// TwinCAT 3 PLC project PLCIO
// ProgramVersion: 3.1.4024.0
// libraries:
//   Tc2_ControllerToolbox, * (Beckhoff Automation GmbH)
//   Tc2_IoFunctions, * (Beckhoff Automation GmbH)
//   Tc2_ModbusRTU, * (Beckhoff Automation GmbH)
//   Tc2_ModbusSrv, * (Beckhoff Automation GmbH)
//   Tc2_SerialCom, * (Beckhoff Automation GmbH)
//   Tc2_Standard, * (Beckhoff Automation GmbH)
//   Tc2_System, * (Beckhoff Automation GmbH)
//   Tc2_TempController, * (Beckhoff Automation GmbH)
//   Tc2_Utilities, * (Beckhoff Automation GmbH)
//   Tc3_EventLogger, * (Beckhoff Automation GmbH)
//   Tc3_Module, * (Beckhoff Automation GmbH)
// project tree:
//   DUTs/ ST_CSV_Record.TcDUT, ST_Recipe1.TcDUT, ST_Array.TcDUT
//   GVLs/ GVL.TcGVL, GVL_CMD.TcGVL (not stored), GVL_COM.TcGVL, GVL_IO.TcGVL (not stored), GVL_OP_A.TcGVL (not stored), GVL_OP_D.TcGVL (not stored), GVL_P2P.TcGVL (not stored), GVL_Recipe.TcGVL
//   / PlcTask.TcTTO, RecipeManager.TcRMO (not stored)
//   POUs/CSV read_write in binary mode/ P_BinaryModeRead.TcPOU, P_BinaryModeWrite.TcPOU
//   POUs/CSV read_write in text mode/ P_TextModeRead.TcPOU, P_TextModeWrite.TcPOU
//   POUs/ Convert2Csv.TcPOU, MAIN.TcPOU, P_ArgToConvExample.TcPOU, P_StringToConvExample.TcPOU, RecipeHandler.TcPOU, TextFieldInputHandler.TcPOU, VisuInit.TcPOU
//   POUs/FunctionBlock/ FB_AI_STATUS_Check.TcPOU, FB_AVG10.TcPOU, FB_DeviationCheck.TcPOU, FB_NoiseCheck.TcPOU, FB_PID.TcPOU, FB_Ramp2.TcPOU, FB_RampControl.TcPOU, FB_Ramp_0.TcPOU, FB_RcpRamp.TcPOU
//   POUs/Function/ F_ET2Sec.TcPOU, F_Int2Real.TcPOU, F_LH_PV.TcPOU, F_LH_SV.TcPOU, F_OPSTATE.TcPOU, F_TB_PV2REAL.TcPOU, F_TB_Rx_BCC.TcPOU, F_TB_SV2STR.TcPOU, F_TB_Tx_BCC.TcPOU
//   POUs/MR_PRG/ P00_Main.TcPOU, P00_OP.TcPOU, P01_Init_N_Retain.TcPOU, P02_Init_MC.TcPOU, P11_Rx_TV.TcPOU, P12_Rx_IH.TcPOU, P13_DI_N_Check.TcPOU, P15_AI.TcPOU, P21_AL_WN.TcPOU, P22_RCP_Ctrl.TcPOU, P24_Rot_Calibration.TcPOU, P25_US_Ctrl.TcPOU, P31_BypassV.TcPOU, P41_DOR_VAC.TcPOU, P41_DOR_VAC_Check.TcPOU, P42_DOR_ATM.TcPOU, P43_SH_UpDw.TcPOU, P49_MO_SRC.TcPOU, P53_DO_VV.TcPOU, P54_DO_ETC.TcPOU, P61_AO.TcPOU, P62_Tx_TV.TcPOU, P63_Tx_IH.TcPOU, REF_P02_KL1501.TcPOU
//   POUs/P02_P2P/ P00_Task_Fast.TcPOU, P02_P2P.TcPOU, P2P_LH.TcPOU, P2P_TB.TcPOU, Task_Fast_LH.TcPOU, Task_Fast_TB.TcPOU
// real-time tasks:
//   TASK PlcTask: cycle T#10ms, priority 20, ADS port 350
//   TASK PlcRecipe: cycle T#10ms, priority 1, ADS port 351

CONFIGURATION PLCIO
    RESOURCE PLC ON TwinCAT3
        TASK PlcTask(INTERVAL := T#10ms, PRIORITY := 20);
        PROGRAM MAIN WITH PlcTask : MAIN;
        PROGRAM RecipeHandler WITH PlcTask : RecipeHandler;
    END_RESOURCE
END_CONFIGURATION

// ---- DUTs/ST_CSV_Record.TcDUT
TYPE ST_CSV_Record :
STRUCT
	sName 	: T_MaxString 	:= '';
	nNumber	: UDINT 		:= 0;
	fPos	: LREAL 		:= 0.0;
	bOP		: BOOL 			:= FALSE;
	sDesc	: STRING(40)	:= '';
	data	: ARRAY[0..7] OF BYTE;
END_STRUCT
END_TYPE

// ---- DUTs/ST_Recipe1.TcDUT
TYPE ST_Recipe1 :
STRUCT
	No    	  :	INT	  ;
	rTime     : INT   ;	
	hTime     : INT   ;	
	rTemp     : INT   ;	
	rPressure : INT   ;	
	sRotation : INT   ;	
	cTemp     : INT   ;	
	Loop      : INT   ;	
	Jump      : INT   ;	
	M01 	  : REAL ;
	M02 	  : REAL ;
	M03 	  : REAL ;
	M04 	  : REAL ;
	M05 	  : REAL ;
	M06 	  : REAL ;
	M07 	  : REAL ;
	M08 	  : REAL ;
	M09 	  : REAL ;
	M10 	  : REAL ;
	M11 	  : REAL ;
	M12 	  : REAL ;
	M13 	  : REAL ;
	M14 	  : REAL ;
	M15 	  : REAL ;
	M16 	  : REAL ;
	M17 	  : REAL ;
	M18 	  : REAL ;
	M19 	  : REAL ;
	E01 	  : REAL ;
	E02 	  : REAL ;
	E03 	  : REAL ;
	E04 	  : REAL ;
	E05 	  : REAL ;
	E06 	  : REAL ;
	E07 	  : REAL ;
	V01 	  : BOOL  ;
	V02 	  : BOOL  ;
	V03 	  : BOOL  ;
	V04 	  : BOOL  ;
	V05 	  : BOOL  ;
	V07 	  : BOOL  ;
	V08 	  : BOOL  ;
	V10 	  : BOOL  ;
	V11 	  : BOOL  ;
	V13 	  : BOOL  ;
	V14 	  : BOOL  ;
	V16 	  : BOOL  ;
	V17 	  : BOOL  ;
	V19 	  : BOOL  ;
	V20 	  : BOOL  ;
	V22 	  : BOOL  ;
	V23 	  : BOOL  ;
	V24 	  : BOOL  ;
	V25 	  : BOOL  ;
	V26 	  : BOOL  ;
	V27 	  : BOOL  ;
	V28 	  : BOOL  ;
	V29 	  : BOOL  ;
	V30 	  : BOOL  ;
	V31 	  : BOOL  ;
	V32 	  : BOOL  ;
END_STRUCT
END_TYPE

// ---- DUTs/ST_Array.TcDUT
TYPE ST_Array :
STRUCT
	IntArr  : ARRAY [0..8] OF INT	  ;
	RealArr  : ARRAY [0..25] OF REAL	  ;
	BoolArr  : ARRAY [0..25] OF BOOL	  ;

END_STRUCT
END_TYPE

// ---- GVLs/GVL.TcGVL
{attribute 'qualified_only'}
VAR_GLOBAL
	EL1088_IN	AT%I*	: BYTE;
	EL2088_OUT	AT%Q*	: BYTE;
	EL3054_IN	AT%I*	: INT;
	EL4024_OUT	AT%Q*	: INT;
	
	gRecipe1 : ST_Recipe1;
	gArray1 : ST_Array;
END_VAR

// ---- GVLs/GVL_COM.TcGVL
//{attribute 'qualified_only'}
VAR_GLOBAL
	
	//NAME -> UPPER CASE
	ON: BOOL := TRUE;
	OFF: BOOL := FALSE;
		
	//Analog Ramp Control	
	RTM_UNIT: TIME;//System Analog Ramping Time unit
	
	s_is_RCP_pause: BOOL;
	s_is_RAMP_stop: BOOL;
	s_is_RAMP_restart: BOOL;

    KL1501_Error: BOOL;//KL1501
	    		
	//Function Execute Bit
	s_EN_EXE_RCP: BOOL;
	s_EN_EXE_DOR_ATM: BOOL;
	s_EN_EXE_DOR_VAC: BOOL;
	s_EN_EXE_ROT_CALI: BOOL;
	
	s_cm_ALL_MC_on: BOOL;
	s_is_All_MC_on: BOOL;
	
	s_en_ROT_JOG: BOOL;
	s_en_ROT_INCH: BOOL;
	s_en_DO_TEST: BOOL;
	
	//P_AL_Rised : BOOL;	
	s_cm_RST: BOOL;	
	s_DOR_CNT: INT;//DOR Alarm check
	s_is_DOR_Broken: BOOL; //IB00_Reactor_Close_Warn : BOOL;

	s_P_RampEN: BOOL;
			
END_VAR

// ---- GVLs/GVL_Recipe.TcGVL
{attribute 'qualified_only'}
VAR_GLOBAL
	No			:	INT;
	rTime		:   INT;
	hTime		:   INT;
	rTemp		:   INT;
	rPressure	:   INT;
	sRotation	:   INT;
	cTemp		:   INT;
	Loop		:   INT; 
	Jump		:   INT; 
	M01         :	REAL;
	M02         :   REAL;
	M03         :   REAL;
	M04         :   REAL;
	M05         :   REAL;
	M06         :   REAL;
	M07         :   REAL;
	M08         :   REAL;
	M09         :   REAL;
	M10         :   REAL;
	M11         :   REAL;
	M12         :   REAL;
	M13         :   REAL;
	M14         :   REAL;
	M15         :   REAL;
	M16         :   REAL;
	M17         :   REAL;
	M18         :   REAL;
	M19         :   REAL;
	E01         :   REAL;
	E02         :   REAL;
	E03         :   REAL;
	E04         :   REAL;
	E05         :   REAL;
	E06         :   REAL;
	E07         :   REAL;
	V01         :   BOOL;
	V02         :   BOOL;
	V03         :   BOOL;
	V04         :   BOOL;
	V05         :   BOOL;
	V07         :   BOOL;
	V08         :   BOOL;
	V10         :   BOOL;
	V11         :   BOOL;
	V13         :   BOOL;
	V14         :   BOOL;
	V16         :   BOOL;
	V17         :   BOOL;
	V19         :   BOOL;
	V20         :   BOOL;
	V22         :   BOOL;
	V23         :   BOOL;
	V24         :   BOOL;
	V25         :   BOOL;
	V26         :   BOOL;
	V27         :   BOOL;
	V28         :   BOOL;
	V29         :   BOOL;
	V30         :   BOOL;
	V31         :   BOOL;
	V32         :   BOOL;

END_VAR

// ---- POUs/MAIN.TcPOU
PROGRAM MAIN
VAR
	plc_state : BOOL;
	plc_array : ARRAY [0..7]  OF BOOL;
	plc_array2 : ARRAY [0..7]  OF BOOL;
	
	p_V05, p_V06: R_TRIG;
	p_V08, p_V09: R_TRIG;
	p_V11, p_V12: R_TRIG;
	p_V14, p_V15: R_TRIG;
	p_V17, p_V18: R_TRIG;
	p_V20, p_V21: R_TRIG;
	
	n_V05, n_V06: F_TRIG;
	n_V08, n_V09: F_TRIG;
	n_V11, n_V12: F_TRIG;
	n_V14, n_V15: F_TRIG;
	n_V17, n_V18: F_TRIG;
	n_V20, n_V21: F_TRIG;
	
	ctime : TIME :=  T#1D14H30M40S500MS;
	lctime : LTIME ;
	cdate : DATE :=  D#2024-07-07;
	str : STRING ;
	wstr : STRING;
	tempstr : STRING;


	OnTimer : TON;
	OffTimer : TOF;
	EnableTimer : BOOL;
	TimerOutPut : BOOL;	
	OnTimerOut : BOOL;
	ReverseSignal : BOOL;
	OffTimerOut : BOOL;
	count : INT;
	el2088_out : BYTE;
	el4024_out : INT;
	el3054_in : INT;
	i : INT;
	j : INT;
	rtime : INT;
	hTime : INT;
	
END_VAR

plc_state := TRUE;

//P00_Main();
p_V05(CLK:= cm_V05); p_V06(CLK:= cm_V06);
p_V08(CLK:= cm_V08); p_V09(CLK:= cm_V09);
p_V11(CLK:= cm_V11); p_V12(CLK:= cm_V12);
p_V14(CLK:= cm_V14); p_V15(CLK:= cm_V15);
p_V17(CLK:= cm_V17); p_V18(CLK:= cm_V18);
p_V20(CLK:= cm_V20); p_V21(CLK:= cm_V21);

n_V05(CLK:= cm_V05); n_V06(CLK:= cm_V06);
n_V08(CLK:= cm_V08); n_V09(CLK:= cm_V09);
n_V11(CLK:= cm_V11); n_V12(CLK:= cm_V12);
n_V14(CLK:= cm_V14); n_V15(CLK:= cm_V15);
n_V17(CLK:= cm_V17); n_V18(CLK:= cm_V18);
n_V20(CLK:= cm_V20); n_V21(CLK:= cm_V21);

IF ing_MAINT = 0 THEN
	
	//interLock Valve Check
	IF p_V05.Q THEN cm_V06 := 1; END_IF  //V05 Open -> V06 Close
	IF n_V05.Q THEN cm_V06 := 0; END_IF	
	IF p_V06.Q THEN cm_V05 := 1; END_IF  //V06 Close -> V05 Open
	IF n_V06.Q THEN cm_V05 := 0; END_IF
		
	IF p_V08.Q THEN cm_V09 := 1; END_IF  //V08 Open -> V09 Close
	IF n_V08.Q THEN cm_V09 := 0; END_IF
	IF p_V09.Q THEN cm_V08 := 1; END_IF  //V09 Close -> V08 Open
	IF n_V09.Q THEN cm_V08 := 0; END_IF
	
	IF p_V11.Q THEN cm_V12 := 1; END_IF  //V11 Open -> V12 Close
	IF n_V11.Q THEN cm_V12 := 0; END_IF
	IF p_V12.Q THEN cm_V11 := 1; END_IF  //V12 Close -> V11 Open
	IF n_V12.Q THEN cm_V11 := 0; END_IF
	
	IF p_V14.Q THEN cm_V15 := 1; END_IF  //V14 Open -> V15 Close
	IF n_V14.Q THEN cm_V15 := 0; END_IF
	IF p_V15.Q THEN cm_V14 := 1; END_IF  //V15 Close -> V14 Open
	IF n_V15.Q THEN cm_V14 := 0; END_IF
	
	IF p_V17.Q THEN cm_V18 := 1; END_IF  //V17 Open -> V18 Close
	IF n_V17.Q THEN cm_V18 := 0; END_IF
	IF p_V18.Q THEN cm_V17 := 1; END_IF  //V18 Close -> V17 Open
	IF n_V18.Q THEN cm_V17 := 0; END_IF
	
	IF p_V20.Q THEN cm_V21 := 1; END_IF  //V20 Open -> V21 Close
	IF n_V20.Q THEN cm_V21 := 0; END_IF
	IF p_V21.Q THEN cm_V20 := 1; END_IF  //V21 Close -> V20 Open
	IF n_V21.Q THEN cm_V20 := 0; END_IF
	
	// Leak Check Valves Off
	cm_V36 := cm_V37 := cm_V38 := cm_V39 := 0;
	cm_V40 := cm_V41 := cm_V42 := cm_V43 := cm_V44 := cm_V45 := 0;
	cm_V46 := cm_V47 := cm_V48 := cm_V49 := cm_V50 := cm_V51 := cm_V52 := 0;
	 
	//Gas Safety Interlock-kjk - Danger Gas Supply Close
	IF is_DOR_VAC_ok = 0 THEN
		IF do_V01 THEN cm_V01 := 0; END_IF//H2 Supply
		IF do_V02 THEN cm_V02 := 0; END_IF//N2 Supply
		IF do_V03 THEN cm_V03 := 0; END_IF//SiH4 Supply
		IF do_V04 THEN cm_V04 := 0; END_IF//NH3 Supply	
	END_IF
 	 
END_IF

do_V01 := cm_V01;
do_V02 := cm_V02;
do_V03 := cm_V03;
do_V04 := cm_V04;
do_V05 := cm_V05;
do_V06 := cm_V06;
do_V07 := cm_V07;
do_V08 := cm_V08;


EnableTimer := TRUE;
IF EnableTimer = TRUE THEN
	OnTimer(IN:=OffTimerOut, Pt:= INT_TO_TIME(1000), Q=>OnTimerOut, ET=>);
	
	IF OnTimerOut = TRUE THEN
		ReverseSignal := FALSE;
		do_V01 := TRUE;
		do_V02 := FALSE;
		do_V03 := TRUE;
		do_V04 := FALSE;
		do_V05 := TRUE;
		do_V06 := FALSE;
		do_V07 := TRUE;
		do_V08 := FALSE;
		tempstr := wstr;

	ELSE
		ReverseSignal := TRUE;
		do_V01 := FALSE;
		do_V02 := TRUE;
		do_V03 := FALSE;
		do_V04 := TRUE;
		do_V05 := FALSE;
		do_V06 := TRUE;
		do_V07 := FALSE;
		do_V08 := TRUE;
		tempstr := str;

	END_IF
	OffTimer(in:=ReverseSignal, pt:= INT_TO_TIME(1000), q=>OffTimerOut,et=>);
	TimerOutput :=OnTimerOut;
	
	el2088_out.0 := do_V01;
	el2088_out.1 := do_V02;
	el2088_out.2 :=	do_V03;
	el2088_out.3 :=	do_V04;
	el2088_out.4 :=	do_V05;
	el2088_out.5 :=	do_V06;
	el2088_out.6 :=	do_V07;
	el2088_out.7 :=	do_V08;
	ctime := ctime + T#10MS;

	
END_IF

cdate :=  D#2024-07-07;
str := 'We are the one, let us heading forwards';

count := count + 1;

GVL.EL4024_OUT := el4024_out;
el3054_in := GVL.EL3054_IN;

EL2088_OUT.0 := do_V01;
EL2088_OUT.1 := do_V02;
EL2088_OUT.2 := do_V03;
EL2088_OUT.3 := do_V04;
EL2088_OUT.4 := do_V05;
EL2088_OUT.5 := do_V06;
EL2088_OUT.6 := do_V07;
EL2088_OUT.7 := do_V08;
plc_array[0] := EL2088_OUT.0;
plc_array[1] := EL2088_OUT.1;
plc_array[2] := EL2088_OUT.2;
plc_array[3] := EL2088_OUT.3;
plc_array[4] := EL2088_OUT.4;
plc_array[5] := EL2088_OUT.5;
plc_array[6] := EL2088_OUT.6;
plc_array[7] := EL2088_OUT.7;

END_PROGRAM

// ---- POUs/RecipeHandler.TcPOU
/// 이 어플리케이션은 ST언어로 RecipeManagement 라이브러리 사용 예제
PROGRAM RecipeHandler
VAR CONSTANT
	AllRecipeDefinitions : ARRAY[0..1] OF STRING := [ 'Recipe1', 'Array1'];
END_VAR
VAR
	initRecipe : BOOL :=TRUE;
	fbFormat : FB_FormatString;

	RecipeManCommands 		: RecipeManCommands; (* Recipe Manager *)
	RecipeDefinition		: IRecipeDefinition2; // current
	
	dwLastError 			: DWORD; (* Error from Recipe Manager *)
	iRecipesCount 			: INT;
	
	sRecipeDef 				: STRING := AllRecipeDefinitions[1]; (* current recipe definition *)
	sRecipe 				: STRING; (*Selected recipe *)
	sRecipeIndex			: INT := 1; // selected recipe index of recipes
	
	xReloadFromFile 		: BOOL; (* Refresh recipes from files *)

	xSaveVariables			: BOOL; // save the variables currently visible in the table to the recipe
	xRefreshRecipes 		: BOOL := False; // refresh the names of the recipes in the currently selected definition
	xReloadValues			: BOOL; // reload the variables and values in the currently selected recipe
	
	xCreateRecipe 			: BOOL; // Creates a new recipe
	xLoadAndWriteRecipe		: BOOL;	
	xDeleteRecipe			: BOOL; // Deletes the selected recipe

	xIsEditingVariable		: BOOL; // signals that one of the textfields where the variable values can be edited is currently being edited
	
	// recipe name을 선택하기 위한 드롭다운
	iRecipeDefinitonNameIndex : INT; // index of the currently selected entry in the Recipe definitions name dropdown
	iPrevRecipeDefinitonNameIndex : INT := -1; // previous index of the currently selected entry in the Recipe definitions name dropdown (to detect refresh needed)
	
	// recipe name들을 표시하기 위한 테이블 작성
	arrRecipeNames 			: ARRAY[0..MAX_TABLE_ROWS-1] OF STRING; // array where the names of the recipes are being stored
	
	iPrevSelectionIndex	 	: INT; // Last selected index of rows
	iRecipeScrollIndex 		: INT; // index showing how far the recipe names table is scrolled
	iPrevScrollIndex 		: INT; // previous value of iRecipeScrollIndex
	iRecipeSelectionIndex 	: INT; // index into the recipe names array
	
	// for the table that displays the variables of a recipe
	arrVariableNames 		: ARRAY[0..(MAX_VARIABLES_TABLE_ROWS-1)] OF STRING; // array where variable names are temporarily stored so they can be displayed
	arrVariableValues 		: ARRAY[0..(MAX_VARIABLES_TABLE_ROWS-1)] OF STRING; // array where variable values are temporarily stored so they can be displayed
	iVariableIndex			: INT; // index into the arrays above which indicates the variable currently being displayed in the first row
	iPrevVariableIndex		: INT; // iVariableIndex from previous call to allow detecting changes
	iVariableCount 			: DINT; // number of variables in the recipe
END_VAR
VAR CONSTANT
	MAX_VARIABLES_TABLE_ROWS 	: INT := 100;
	MAX_TABLE_ROWS 				: INT := 100;
END_VAR
VAR_OUTPUT
	hasError : BOOL; // if there is some sort of internal error
END_VAR
VAR_TEMP
	i : INT; // loop index
END_VAR

hasError := FALSE;

IF initRecipe THEN
	iRecipesCount := RecipeManCommands.GetRecipeCount(sRecipeDef);

	FOR i := 1 TO iRecipesCount DO
		xCreateRecipe := TRUE;
		fbFormat(sFormat := 'r%d', arg1 := F_INT(sRecipeIndex), sOut => sRecipe);
		IF xCreateRecipe THEN
			IF RecipeManCommands.CreateRecipe(sRecipeDef, sRecipe) <> ERR_OK THEN
				hasError := TRUE;
				RETURN;
			END_IF
		//	xRefreshRecipes := TRUE;
		END_IF
	
	END_FOR
	xCreateRecipe := FALSE;
	initRecipe := FALSE;	
END_IF


//// check if one of the variables has been edited
//// NOTE: to prevent bad timing effects this PRG should be executed in VisuTask
//IF xIsEditingVariable AND VisuInit.TFHandler.finishedEdit (* this must be manually set to false when the edit begins*) THEN
//	VisuInit.TFHandler.finishedEdit := FALSE;
//	xSaveVariables := TRUE;
//	xIsEditingVariable := FALSE;
//END_IF

//(* Set the edited values into the recipe *)
//IF xSaveVariables THEN
////	RecipeManCommands.SetRecipeValues(sRecipeDef, sRecipe, ADR(arrVariableValues), MAX_VARIABLES_TABLE_ROWS, iVariableIndex);
//	RecipeManCommands.SaveRecipe(sRecipeDef, sRecipe);
//	xSaveVariables := FALSE;
//END_IF

//// get current recipe definition name from visu
//IF iPrevRecipeDefinitonNameIndex <> iRecipeDefinitonNameIndex THEN
//	sRecipeDef := AllRecipeDefinitions[iRecipeDefinitonNameIndex];
//	xRefreshRecipes := TRUE;
//	xReloadValues := TRUE;
//END_IF
//iPrevRecipeDefinitonNameIndex := iRecipeDefinitonNameIndex;

//(* Load the list of the recipes in the selected recipe definition*)
//IF xRefreshRecipes THEN
//	(* Save the number of recipes in the specified recipe definition in a global variable.*)
//	iRecipesCount := RecipeManCommands.GetRecipeCount(sRecipeDef);
//	(* Empty all arrays *)
//	FOR i := 0 TO MAX_TABLE_ROWS DO
//		arrRecipeNames[i] := '';
//		arrVariableNames[i] := '';
//		arrVariableValues[i] := '';
//	END_FOR
//	(* save all recipe names of one recipe definition in an array *)
//	RecipeManCommands.GetRecipeNames(sRecipeDef, ADR(arrRecipeNames), 10, iRecipeScrollIndex);
//	xReloadValues := TRUE;
//	xRefreshRecipes := FALSE;
//END_IF

//dwLastError := RecipeManCommands.GetLastError();

//(* Scroll position of the recipe list has changed. *)
//IF iRecipeScrollIndex <> iPrevScrollIndex THEN
//	RecipeManCommands.GetRecipeNames(sRecipeDef, ADR(arrRecipeNames), 10, iRecipeScrollIndex);
//	iPrevScrollIndex := iRecipeScrollIndex;
//END_IF

//(* Selection of the current recipe has changed *)
//IF iRecipeSelectionIndex <> iPrevSelectionIndex OR iPrevVariableIndex <> iVariableIndex OR xReloadValues THEN
//	iPrevSelectionIndex := iRecipeSelectionIndex;
//	iPrevVariableIndex := iVariableIndex;

//	(* Get the selected recipe name *)
//	// the (iRecipeSelectionIndex - iRecipeScrollIndex) thing is needed so we get the index into the names array
//	IF (iRecipeSelectionIndex - iRecipeScrollIndex) >= 0 AND (iRecipeSelectionIndex - iRecipeScrollIndex) < MAX_TABLE_ROWS THEN
//		sRecipe := arrRecipeNames[(iRecipeSelectionIndex - iRecipeScrollIndex)];
//	END_IF
	
//	// update number of variables for the new recipe
//	iRecipesCount := RecipeManCommands.GetRecipeCount(sRecipeDef); // this makes sure that _RecipeDefinition is set to the one we want
//	IF __QUERYINTERFACE(RecipeManCommands._RecipeDefinition, RecipeDefinition) THEN
//		{analysis -46} // RecipeDefinition is definitly initialized
//		iVariableCount := RecipeDefinition.GetRecipeVariableCount();
//		{analysis +46}
//	ELSE
//		iVariableCount := 999; // set a default if we cannot determine it
//	END_IF

//	IF RecipeManCommands.GetRecipeValues(sRecipeDef, sRecipe, ADR(arrVariableValues), MAX_VARIABLES_TABLE_ROWS, iVariableIndex, 80) <> ERR_OK OR_ELSE
//		LEN(sRecipe) = 0 (* for empty string ERR_OK is returned, so we need to manually check for that *)
//	THEN	
//		// error while loading, blank out the column
//		FOR i := 0 TO 	MAX_VARIABLES_TABLE_ROWS - 1 DO
//			arrVariableValues[i] := 'xxx';
//		END_FOR
//	END_IF
//	IF RecipeManCommands.GetRecipeVariableNames(sRecipeDef, sRecipe, ADR(arrVariableNames), MAX_VARIABLES_TABLE_ROWS, iVariableIndex) <> ERR_OK THEN
//		// error while loading, blank out the column
//		FOR i := 0 TO 	MAX_VARIABLES_TABLE_ROWS - 1 DO
//			arrVariableValues[i] := 'yyy';
//		END_FOR
//	END_IF

//	xReloadValues := FALSE;
//END_IF

(* Reload the recipe list from the file system *)
//IF xReloadFromFile THEN
//	IF RecipeManCommands.ReloadRecipes(sRecipeDef) <> ERR_OK THEN
//		hasError := TRUE;
//		RETURN;
//	END_IF
////	xRefreshRecipes := TRUE;
////	xReloadFromFile := FALSE;
//END_IF

IF xCreateRecipe THEN
	IF RecipeManCommands.CreateRecipe(sRecipeDef, sRecipe) <> ERR_OK THEN
		hasError := TRUE;
		RETURN;
	END_IF
	xCreateRecipe := FALSE;	
//	xRefreshRecipes := TRUE;
END_IF

IF xLoadAndWriteRecipe THEN
	fbFormat(sFormat := 'r%d', arg1 := F_INT(sRecipeIndex), sOut => sRecipe);

	IF RecipeManCommands.LoadandWriteRecipe(sRecipeDef, sRecipe) <> ERR_OK THEN
		hasError := TRUE;
		RETURN;
	END_IF
//	xRefreshRecipes := TRUE;
//	xReloadFromFile := FALSE;
END_IF

IF xDeleteRecipe THEN
	IF RecipeManCommands.DeleteRecipe(sRecipeDef, sRecipe) <> ERR_OK THEN
		hasError := TRUE;
		RETURN;
	END_IF
//	xRefreshRecipes := TRUE;
END_IF

END_PROGRAM

// ---- POUs/CSV read_write in binary mode/P_BinaryModeRead.TcPOU
(* Reading of CSV file in binary mode. Field values may contain non-printing control characters (binary data or special characters like line feed, carriage return or quotation mark...). *)
PROGRAM P_BinaryModeRead
VAR
	bRead		: BOOL := FALSE;(* Rising edge starts program execution *)
	sNetId		: T_AmsNetId := '';	(* TwinCAT system network address *)
	sFileName	: T_MaxString := 'C:\Temp\BinaryModeGen.csv';(* CSV source file path and name *)
	bBusy		: BOOL;
	bError		: BOOL;
	nErrId		: UDINT;
	nRow	 	: UDINT 	:= 0;(* Row number (record) *)
	nColumn		: UDINT 	:= 0;(* Column number (record field) *)
	cbDone		: UDINT 	:= 0;(* Counts allready parsed data bytes *)
	hFile		: UINT		:= 0;(* File handle of the source file *)
	step		: DWORD 	:= 0;
	fbFileOpen	: FB_FileOpen;(* Opens file *)
	fbFileClose	: FB_FileClose;(* Closes file *)
	fbFileRead	: FB_FileRead;(* Writes binary data *)
	fbReader	: FB_CSVMemBufferReader;(* Helper function block used to parse CSV data bytes *)

	record		: ARRAY[0..1024] OF BYTE;(* Binary row data buffer. The size of this buffer have to be > length of longest record line + 2 (CRLF)  *)
	cbRecord	: UDINT := 0;(* Number of bytes in row buffer *)
	cbField		: UDINT;(* Number of bytes in field buffer *)

	database	: ARRAY[0..MAX_CSV_ROWS ] OF ST_CSV_Record;(* Target PLC database *)
END_VAR

CASE step OF
	0:	(* Wait for rising edge at bRead variable *)
		IF bRead THEN
			bRead 	:= FALSE;
			bBusy 	:= TRUE;
			bError	:= FALSE;
			nErrId	:= 0;
			hFile	:= 0;
			nRow	:= 0;
			nColumn	:= 0;
			cbRecord:= 0;
			cbDone 	:= 0;
			step 	:= 1;
		END_IF

	1:	(* Open source file *)
		fbFileOpen(  bExecute := FALSE  );
		fbFileOpen( sNetId := sNetId, sPathName := sFileName, nMode := FOPEN_MODEREAD OR FOPEN_MODEBINARY,(* Open file in BINARY mode! *)
					ePath := PATH_GENERIC, bExecute := TRUE );
		step := 2;

	2:(* Wait until open not busy *)
		fbFileOpen( bExecute := FALSE, bError => bError, nErrID => nErrID, hFile => hFile );
		IF NOT fbFileOpen.bBusy THEN
			IF NOT fbFileOpen.bError THEN
				step := 3;
			ELSE(* Error: file not found? *)
				step := 100;
			END_IF
		END_IF

	3:	(* Read data bytes from file *)
		fbFileRead( bExecute := FALSE );
		fbFileRead( sNetId := sNetId, hFile := hFile, pReadBuff := ADR( record[ cbRecord ] ), cbReadLen := SIZEOF( record ) - cbRecord, bExecute :=TRUE );
		step := 4;

	4:(* Wait until read not busy *)
		fbFileRead( bExecute := FALSE, bError => bError, nErrID => nErrID );
		IF NOT fbFileRead.bBusy THEN
			IF NOT fbFileRead.bError THEN
				IF fbFileRead.bEOF THEN
					step := 10;(* End of file reached => Close source file *)
				ELSE
					cbRecord := cbRecord + fbFileRead.cbRead;(* Recalculate the new size of data buffer *)
					step := 5;(* Parse binary data *)
				END_IF
			ELSE(* Error *)
				step := 100;
			END_IF
		END_IF

	5:(* Parse binary data *)
		cbDone := 0;(* Reset number of parsed data bytes *)
		fbReader.eCmd := eEnumCmd_First;(* Read first field value *)
		REPEAT
			fbReader( pBuffer := ADR( record ), cbBuffer := cbRecord );
			IF fbReader.bOk THEN
				fbReader.eCmd := eEnumCmd_Next;(* Read next field value *)
				cbDone := cbDone + fbReader.cbRead;(* Count the number of successfully parsed data bytes *)

				IF ( nRow <= MAX_CSV_ROWS ) THEN
					(* Convert every CSV data field to PLC data field format *)
					CASE nColumn OF
						0:(* sName : T_MaxString *)
							cbField := CSVFIELD_TO_ARG( fbReader.pValue, fbReader.cbValue,  TRUE, F_STRING( database[nRow].sName ) );
						1:(* nNumber : UDINT *)
							cbField := CSVFIELD_TO_ARG( fbReader.pValue, fbReader.cbValue,  TRUE, F_UDINT( database[nRow].nNumber ) );
						2:(* fPos : LREAL *)
							cbField := CSVFIELD_TO_ARG( fbReader.pValue, fbReader.cbValue,  TRUE, F_LREAL( database[nRow].fPos ) );
						3:(* bOP : BOOL *)
							cbField := CSVFIELD_TO_ARG( fbReader.pValue, fbReader.cbValue,  TRUE, F_BOOL( database[nRow].bOP ) );
						4:(* sDesc : STRING(40) *)
							cbField := CSVFIELD_TO_ARG( fbReader.pValue, fbReader.cbValue,  TRUE, F_BIGTYPE( ADR( database[nRow].sDesc ), SIZEOF( database[nRow].sDesc ) ) );
						5:(* data : ARRAY[0..7] OF BYTE *)
							cbField := CSVFIELD_TO_ARG( fbReader.pValue, fbReader.cbValue,  TRUE, F_BIGTYPE( ADR( database[nRow].data ), SIZEOF( database[nRow].data ) ) );
					ELSE
						;
					END_CASE
				END_IF

				nColumn := nColumn + 1;(* Increment number of read columns *)
				IF fbReader.bCRLF THEN(* CRLF == TRUE => End of reacord reached *)
					nRow 		:= nRow + 1;(* Increment number of read records *)
					nColumn 	:= 0;(* Reset number of columns *)
				END_IF

			ELSE(* Error: End of buffer reached or all fields parsed *)
				cbRecord := MEMMOVE( ADR( record ), ADR( record[ cbDone ] ), cbRecord - cbDone );(* Shift left the remaining (not allready read) data bytes *)
				step := 3;(* Read new data bytes *)
			END_IF
		UNTIL NOT fbReader.bOk
		END_REPEAT

	10:	(* Close source file *)
		fbFileClose( bExecute := FALSE );
		fbFileClose( sNetId := sNetId, hFile := hFile, bExecute := TRUE );
		step := 11;

	11:(* Wait until close not busy *)
		fbFileClose( bExecute := FALSE, bError => bError, nErrID => nErrID );
		IF ( NOT fbFileClose.bBusy ) THEN
			hFile := 0;
			step := 100;
		END_IF

	100: (* Error or ready step => cleanup *)
		IF ( hFile <> 0 ) THEN
			step := 10; (* Close the source file *)
		ELSE
			bBusy := FALSE;
			step := 0;	(* Ready *)
		END_IF

END_CASE

END_PROGRAM

// ---- POUs/CSV read_write in binary mode/P_BinaryModeWrite.TcPOU
(* Writing of CSV file in binary mode. Field values may contain non-printing control characters (binary data or special characters like line feed, carriage return or quotation mark...). *)
PROGRAM P_BinaryModeWrite
VAR
	bWrite		: BOOL := FALSE;(* Rising edge starts program execution *)
	sNetId		: T_AmsNetId := '';	(* TwinCAT system network address *)
	sFileName	: T_MaxString := 'C:\Temp\BinaryModeGen.csv';(* CSV destination file path and name *)
	bBusy		: BOOL;
	bError		: BOOL;
	nErrId		: UDINT;
	nRow	 	: UDINT 	:= 0;(* Row number (record) *)
	nColumn		: UDINT 	:= 0;(* Column number (record field) *)
	hFile		: UINT		:= 0;(* File handle of the source file *)
	step		: DWORD 	:= 0;

	fbFileOpen	: FB_FileOpen;(* Opens file *)
	fbFileClose	: FB_FileClose;(* Closes file *)
	fbFileWrite	: FB_FileWrite;(* Reads binary data *)
	fbWriter	: FB_CSVMemBufferWriter;(* Helper function block used to create CSV data bytes *)

	record		: ARRAY[0..1024] OF BYTE;(* Binary (row) data buffer. The size of this buffer have to be > length of longest record line + 2 (CRLF)  *)
	cbRecord	: UDINT := 0;(* Number of bytes in row buffer *)
	field		: ARRAY[0..MAX_CSV_FIELD_LENGTH] OF BYTE;(* Binary (field) data buffer. The size of this buffer have to be > length of the longest field *)
	cbField		: UDINT;(* Number of bytes in field buffer *)

	database 	: ARRAY[0..MAX_CSV_ROWS] OF ST_CSV_Record :=[ (* Source PLC database *)
	( sName := '0_0', nNumber := 1,  fPos := 0.1, bOp := FALSE, sDesc := 'Module: "ADX1", ID: $01;$R$L', data 	:=[ 0,1,2,3,4,5,6,7] ),
	( sName := '1_0', nNumber := 2,  fPos := 0.2, bOp := TRUE, 	sDesc := 'Module: "BDX2", ID: $02;$R$L', data 	:=[ 8,9,10,11,12,13,14,15] ),
	( sName := '2_0', nNumber := 3,  fPos := 0.3, bOp := FALSE, sDesc := 'Module: "CDX3", ID: $03;$R$L', data 	:=[ 16,17,18,19,20,21,22,23] ),
	( sName := '3_0', nNumber := 4,  fPos := 0.4, bOp := TRUE, 	sDesc := 'Module: "DDX4", ID: $04;$R$L', data 	:=[ 24,25,26,27,28,29,30,31] ),
	( sName := '4_0', nNumber := 5,  fPos := 0.5, bOp := FALSE, sDesc := 'Module: "EDX5", ID: $05;$R$L', data 	:=[ 32,33,34,35,36,37,38,39] ),
	( sName := '5_0', nNumber := 6,  fPos := 0.6, bOp := TRUE, 	sDesc := 'Module: "FDX6", ID: $06;$R$L', data 	:=[ 40,41,42,43,44,45,46,47] )];
END_VAR

CASE step OF
	0:	(* Wait for rising edge at bWrite variable *)
		IF bWrite THEN
			bWrite 	:= FALSE;
			bBusy 	:= TRUE;
			bError	:= FALSE;
			nErrId	:= 0;
			hFile	:= 0;
			nRow	:= 0;
			nColumn := 0;
			step 	:= 1;
		END_IF

	1:	(* Open source file *)
		fbFileOpen( bExecute := FALSE  );
		fbFileOpen( sNetId := sNetId, sPathName := sFileName, nMode := FOPEN_MODEWRITE OR FOPEN_MODEBINARY, (* Open file in BINARY mode! *)
					ePath := PATH_GENERIC, bExecute := TRUE );
		step := 2;

	2:(* Wait until open not busy *)
		fbFileOpen( bExecute := FALSE, bError => bError, nErrID => nErrID, hFile => hFile );
		IF NOT fbFileOpen.bBusy THEN
			IF NOT fbFileOpen.bError THEN
				step := 3;
			ELSE(* Error: file not found? *)
				step := 100;
			END_IF
		END_IF

	3:(* Convert one PLC record to CSV format *)
		cbRecord := 0;
		fbWriter.eCmd := eEnumCmd_First;(* Write first field value *)
		IF nRow <= MAX_CSV_ROWS THEN

			(* Convert every PLC data field to the CSV data field format *)
			FOR nColumn := 0 TO MAX_CSV_COLUMNS BY 1 DO

				cbField := 0;(* Reset *)
				CASE nColumn OF
					0:(* sName : T_MaxString *)
						cbField := ARG_TO_CSVFIELD( F_STRING( database[ nRow ].sName ), TRUE, ADR( field ), SIZEOF( field ) );
					1:(* nNumber : UDINT *)
						cbField := ARG_TO_CSVFIELD( F_UDINT( database[ nRow ].nNumber ), TRUE, ADR( field ), SIZEOF( field ) );
					2:(* fPos : LREAL *)
						cbField := ARG_TO_CSVFIELD( F_LREAL( database[ nRow ].fPos ), TRUE, ADR( field ), SIZEOF( field ) );
					3:(* bOP : BOOL  *)
						cbField := ARG_TO_CSVFIELD( F_BOOL( database[ nRow ].bOP ), TRUE, ADR( field ), SIZEOF( field ) );
					4:(* sDesc : STRING(40) *)
						cbField := ARG_TO_CSVFIELD( F_BIGTYPE( ADR( database[ nRow ].sDesc ), INT_TO_DWORD(LEN( database[ nRow ].sDesc ) ) ), TRUE, ADR( field ), SIZEOF( field ) );
					5:(* data :ARRAY[0..7] OF BYTE *)
						cbField := ARG_TO_CSVFIELD( F_BIGTYPE( ADR( database[ nRow ].data ), SIZEOF( database[ nRow ].data ) ), TRUE, ADR( field ), SIZEOF( field ) );
				ELSE
					;
				END_CASE

				IF cbField > 0 THEN
					(* Add new field to the record buffer *)
					fbWriter( 	pBuffer := ADR( record ), cbBuffer := SIZEOF( record ), putValue :='',  pValue := ADR( field ), cbValue := cbField,
								bCRLF := ( nColumn = MAX_CSV_COLUMNS ) );(* bCRLF == TRUE => Write CRLF after the last field value *)
					IF fbWriter.bOk THEN
						fbWriter.eCmd 	:= eEnumCmd_Next;(* Write next field value *)
						cbRecord 		:= cbRecord + fbWriter.cbWrite;(* Calculate the new record size *)
					ELSE(* Error *)
						step := 100;
						RETURN;
					END_IF
				END_IF

			END_FOR(* FOR nColumn := 0... *)

			nRow := nRow + 1;(* Increment number of created records (rows) *)
			step := 4;(* Write record to the file *)

		ELSE(* All rows written => Close file *)
			step := 10;
		END_IF


	4:	(* Write record to file *)
		fbFileWrite( bExecute := FALSE );
		fbFileWrite( sNetId := sNetId, hFile := hFile, pWriteBuff := ADR( record ), cbWriteLen := cbRecord, bExecute := TRUE );
		step := 5;

	5:(* Wait until write not busy *)
		fbFileWrite( bExecute := FALSE, bError => bError, nErrID => nErrID );
		IF NOT fbFileWrite.bBusy THEN
			IF NOT fbFileWrite.bError THEN
				step := 3;(* Write next record *)
			ELSE(* Error *)
				step := 100;
			END_IF
		END_IF

	10:	(* Close source file *)
		fbFileClose( bExecute := FALSE );
		fbFileClose( sNetId := sNetId, hFile := hFile, bExecute := TRUE );
		step := 11;

	11:(* Wait until close not busy *)
		fbFileClose( bExecute := FALSE, bError => bError, nErrID => nErrID );
		IF ( NOT fbFileClose.bBusy ) THEN
			hFile := 0;
			step := 100;
		END_IF

	100: (* Error or ready step => cleanup *)
		IF ( hFile <> 0 ) THEN
			step := 10; (* Close the source file *)
		ELSE
			bBusy := FALSE;
			step := 0;	(* Ready *)
		END_IF

END_CASE

END_PROGRAM

// ---- POUs/CSV read_write in text mode/P_TextModeRead.TcPOU
(* Reading of CSV file in text mode. None of the field value is containing any non-printing control characters like line feed, carriage return, quotation marks, semicolon... *)
PROGRAM P_TextModeRead
VAR
	bRead			: BOOL := FALSE;(* Rising edge starts program execution *)
	sNetId			: T_AmsNetId := '';	(* TwinCAT system network address *)
	sFileName		: T_MaxString := 'D:\study\TwincatProj\csvdata\TextModeGen.csv';(* CSV source file path and name *)
	sCSVLine		: T_MaxString := '';(* Single CSV text line (row, record), we are using string as record buffer (your are able to see read fields)  *)
	sCSVField		: T_MaxString := '';(* Single CSV field value (column, record field) *)
	bBusy			: BOOL;
	bError			: BOOL;
	nErrId			: UDINT;
	nRow	 		: UDINT 	:= 0;(* Row number (record) *)
	nColumn			: UDINT 	:= 0;(* Column number (record field) *)
	hFile			: UINT		:= 0;(* File handle of the source file *)
	step			: DWORD 	:= 0;
	fbFileOpen		: FB_FileOpen;(* Opens file *)
	fbFileClose		: FB_FileClose;(* Closes file *)
	fbFileGets		: FB_FileGets;(* Reads one record (line) *)
	fbReader		: FB_CSVMemBufferReader;(* Helper function block used to parse CSV data bytes (single record line) *)

	database		: ARRAY[0..MAX_CSV_ROWS, 0..MAX_CSV_COLUMNS ] OF STRING(MAX_CSV_FIELD_LENGTH);(* Target PLC database *)
END_VAR

CASE step OF
	0:	(* Wait for rising edge at bRead variable *)
		IF bRead THEN
			bRead 	:= FALSE;
			bBusy 	:= TRUE;
			bError	:= FALSE;
			nErrId	:= 0;
			hFile	:= 0;
			nRow	:= 0;
			nColumn	:= 0;
			MEMSET( ADR( database ), 0, SIZEOF( database ) );
			step 		:= 1;
		END_IF

	1:	(* Open source file *)
		fbFileOpen(  bExecute := FALSE  );
		fbFileOpen( sNetId := sNetId, sPathName := sFileName, nMode := FOPEN_MODEREAD OR FOPEN_MODETEXT,(* Open file in TEXT mode! *)
					ePath := PATH_GENERIC, bExecute := TRUE );
		step := 2;

	2:(* Wait until open not busy *)
		fbFileOpen( bExecute := FALSE, bError => bError, nErrID => nErrID, hFile => hFile );
		IF NOT fbFileOpen.bBusy THEN
			IF NOT fbFileOpen.bError THEN
				step := 3;
			ELSE(* Error: file not found? *)
				step := 100;
			END_IF
		END_IF

	3:	(* Read single line (record) *)
		fbFileGets( bExecute := FALSE );
		fbFileGets( sNetId := sNetId, hFile := hFile, bExecute := TRUE );
		step := 4;

	4:(* Wait until read not busy *)
		fbFileGets( bExecute := FALSE, bError => bError, nErrID => nErrID, sLine => sCSVLine );
		IF NOT fbFileGets.bBusy THEN
			IF NOT fbFileGets.bError THEN
				IF fbFileGets.bEOF THEN
					step := 10;(* End of file reached => Close source file *)
				ELSE

					(* FB_FileGets returns text line without the CR (carriage return) character.
					We have to restore the CR character (replace the $L character with $R$L characters) *)
					IF RIGHT( sCSVLine, 1 ) = '$L' THEN
						sCSVLine := REPLACE( sCSVLine, '$R$L', 2, LEN( sCSVLine ) );
					END_IF

					step := 5;
				END_IF
			ELSE(* Error *)
				step := 100;
			END_IF
		END_IF

	5:(* Parse single line (record) *)
		fbReader.eCmd := eEnumCmd_First;(* Read first field value *)
		REPEAT
			fbReader( pBuffer := ADR( sCSVLine ), cbBuffer := SIZEOF( sCSVLine ), getValue => sCSVField );
			IF fbReader.bOk THEN
				fbReader.eCmd := eEnumCmd_Next;(* Read next field value *)

				IF ( nRow <= MAX_CSV_ROWS ) THEN
					IF ( nColumn <= MAX_CSV_COLUMNS ) THEN
						database[nRow, nColumn] := CSVFIELD_TO_STRING( sCSVField, FALSE );(* TODO: Save or use the field value in your application *)
					END_IF
				END_IF

				nColumn := nColumn + 1;(* Increment number of read columns *)
				IF fbReader.bCRLF THEN(* CRLF == TRUE => End of reacord reached *)
					nRow 		:= nRow + 1;(* Increment number of read records *)
					nColumn 	:= 0;(* Reset number of columns *)
				END_IF

			ELSE(* Error: End of record reached or all fields read *)
				step := 3;(* Try to read next line *)
			END_IF
		UNTIL NOT fbReader.bOk
		END_REPEAT

	10:	(* Close source file *)
		fbFileClose( bExecute := FALSE );
		fbFileClose( sNetId := sNetId, hFile := hFile, bExecute := TRUE );
		step := 11;

	11:(* Wait until close not busy *)
		fbFileClose( bExecute := FALSE, bError => bError, nErrID => nErrID );
		IF ( NOT fbFileClose.bBusy ) THEN
			hFile := 0;
			step := 100;
		END_IF

	100: (* Error or ready step => cleanup *)
		IF ( hFile <> 0 ) THEN
			step := 10; (* Close the source file *)
		ELSE
			bBusy := FALSE;
			step := 0;	(* Ready *)
		END_IF

END_CASE

DB.iDataFromCSVINT:= STRING_TO_INT(database[2,2]);
DB.rDataFromCSVREAL:= STRING_TO_REAL(database[3,2]);

END_PROGRAM

// ---- POUs/CSV read_write in text mode/P_TextModeWrite.TcPOU
(* Writing of CSV file in text mode. None of the field value is containing any non-printing control characters like line feed, carriage return, quotation marks, semicolon... *)
PROGRAM P_TextModeWrite
VAR
	bWrite			: BOOL := FALSE;(* Rising edge starts program execution *)
	sNetId			: T_AmsNetId := '';	(* TwinCAT system network address *)
	sFileName		: T_MaxString := 'D:\study\TwincatProj\csvdata\TextModeGen.csv';(* CSV destination file path and name *)
	sCSVLine		: T_MaxString := '';(* Single CSV text line (row, record), we are using string as record buffer (your are able to see created fields) *)
	sCSVField		: T_MaxString := '';(* Single CSV field value (column, record field) *)
	bBusy			: BOOL;
	bError			: BOOL;
	nErrId			: UDINT;
	nRow	 		: UDINT 	:= 0;(* Row number (record) *)
	nColumn			: UDINT 	:= 0;(* Column number (record field) *)
	hFile			: UINT		:= 0;(* File handle of the source file *)
	step			: DWORD 	:= 0;
	fbFileOpen		: FB_FileOpen;(* Opens file *)
	fbFileClose		: FB_FileClose;(* Closes file *)
	fbFilePuts		: FB_FilePuts;(* Writes one record (line) *)
	fbWriter		: FB_CSVMemBufferWriter;(* Helper function block used to create CSV data bytes (single record line) *)

	database		: ARRAY[0..MAX_CSV_ROWS, 0..MAX_CSV_COLUMNS ] OF STRING(MAX_CSV_FIELD_LENGTH) :=[ (* Source PLC database *)
	'0_0', '0_1', '0_2', '0_3', '0_4', '0_5',
	'1_0', '1_1', '1_2', '1_3', '1_4', '1_5',
	'2_0', '2_1', '2_2', '2_3', '2_4', '2_5',
	'3_0', '3_1', '3_2', '3_3', '3_4', '3_5',
	'4_0', '4_1', '4_2', '4_3', '4_4', '4_5',
	'5_0', '5_1', '5_2', '5_3', '5_4', '5_5'];

END_VAR

CASE step OF
	0:	(* Wait for rising edge at bWrite variable *)
		IF bWrite THEN
			bWrite 	:= FALSE;
			bBusy 	:= TRUE;
			bError	:= FALSE;
			nErrId	:= 0;
			hFile	:= 0;
			nRow	:= 0;
			nColumn	:= 0;
			step 	:= 1;
		END_IF

	1:	(* Open source file *)
		fbFileOpen(  bExecute := FALSE  );
		fbFileOpen( sNetId := sNetId, sPathName := sFileName, nMode := FOPEN_MODEWRITE OR FOPEN_MODETEXT,(* Open file in TEXT mode! *)
					ePath := PATH_GENERIC, bExecute := TRUE );
		step := 2;

	2:(* Wait until open not busy *)
		fbFileOpen( bExecute := FALSE, bError => bError, nErrID => nErrID, hFile => hFile );
		IF NOT fbFileOpen.bBusy THEN
			IF NOT fbFileOpen.bError THEN
				step := 3;
			ELSE(* Error: file not found? *)
				step := 100;
			END_IF
		END_IF

	3:(* Convert one PLC record to CSV format *)
		sCSVLine := '';
		fbWriter.eCmd := eEnumCmd_First;(* Write first field value *)
		IF nRow <= MAX_CSV_ROWS THEN

			FOR nColumn := 0 TO MAX_CSV_COLUMNS BY 1 DO

				sCSVField := STRING_TO_CSVFIELD( database[ nRow, nColumn ], FALSE );(* TODO: Get field value from your application *)

				(* Add new field to the record buffer *)
				fbWriter( 	pBuffer := ADR( sCSVLine ), cbBuffer := SIZEOF( sCSVLine ) - 1, putValue := sCSVField, pValue := 0, cbValue := 0,
							bCRLF := ( nColumn = MAX_CSV_COLUMNS ) );(* bCRLF == TRUE => Write CRLF after the last field value *)
				IF fbWriter.bOk THEN
					fbWriter.eCmd := eEnumCmd_Next;(* Write next field value *)
				ELSE(* Error *)
					step := 100;
					RETURN;
				END_IF

			END_FOR(* FOR nColumn := 0... *)

			(* FB_FilePuts adds allready CR (carriage return) to the written line.
			We have to replace the $R$L characters with $L character to avoid double CR. *)
			IF RIGHT( sCSVLine, 2 ) = '$R$L' THEN
				sCSVLine := REPLACE( sCSVLine, '$L', 2, LEN( sCSVLine ) - 1 );
			END_IF

			nRow := nRow + 1;(* Increment number of created records (rows) *)
			step := 4;(* Write record to the file *)

		ELSE(* All rows written => Close file *)
			step := 10;
		END_IF

	4:	(* Write single text line *)
		fbFilePuts( bExecute := FALSE );
		fbFilePuts( sNetId := sNetId, hFile := hFile, sLine := sCSVLine, bExecute := TRUE );
		step := 5;

	5:(* Wait until write not busy *)
		fbFilePuts( bExecute := FALSE, bError => bError, nErrID => nErrID );
		IF NOT fbFilePuts.bBusy THEN
			IF NOT fbFilePuts.bError THEN
				step := 3;(* Write next record *)
			ELSE(* Error *)
				step := 100;
			END_IF
		END_IF

	10:	(* Close source file *)
		fbFileClose( bExecute := FALSE );
		fbFileClose( sNetId := sNetId, hFile := hFile, bExecute := TRUE );
		step := 11;

	11:(* Wait until close not busy *)
		fbFileClose( bExecute := FALSE, bError => bError, nErrID => nErrID );
		IF ( NOT fbFileClose.bBusy ) THEN
			hFile := 0;
			step := 100;
		END_IF

	100: (* Error or ready step => cleanup *)
		IF ( hFile <> 0 ) THEN
			step := 10; (* Close the source file *)
		ELSE
			bBusy := FALSE;
			step := 0;	(* Ready *)
		END_IF

END_CASE


database[1,0] := INT_TO_STRING(DB.iDataToCSVINT);
database[2,0] := REAL_TO_STRING(db.rDataToCSVREAL);

END_PROGRAM

// ---- POUs/Convert2Csv.TcPOU
PROGRAM Convert2Csv
VAR
		(* In USA/UK the CSV field separator is a comma.
	In Germany and some other European countries the CSV field separator is a semicolon. *)
	bChangeSeparatorToComma	: BOOL := TRUE;
END_VAR

IF bChangeSeparatorToComma THEN
	DEFAULT_CSV_FIELD_SEP := 16#2C;(* Comma ASCII code *)
ELSE
	DEFAULT_CSV_FIELD_SEP := 16#3B;(* Semicolon ASCII code *)
END_IF

P_TextModeRead();(* This sample program opens and reads CSV file in text mode *)

P_TextModeWrite();(* This sample program opens and writes CSV file in text mode *)

P_BinaryModeRead();(* This sample program opens and reads CSV file in binary mode *)

P_BinaryModeWrite();(* This sample program opens and writes CSV file in binary mode *)

P_ArgToConvExample();(* This sample program shows the usage of the ARG_TO_CSVFIELD and CSVFILED_TO_ARG conversion functions *)

P_StringToConvExample();(* This sample program shows the usage of the STRING_TO_CSVFIELD and CSVFIELD_TO_STRING conversion functions *)

END_PROGRAM

// ---- POUs/P_ArgToConvExample.TcPOU
PROGRAM P_ArgToConvExample
VAR
	(* PLC data to be converted to or from CSV format *)
	bOperating	: BOOL := TRUE;
	fAxPos		: LREAL := 12.2;
	nCounter 	: UDINT := 7;
	sName		: T_MaxString := 'Module: "XAF", $04$05, 20';
	binData		: ARRAY[0..9] OF BYTE :=[ 0, 1, 2, 3, 4, 5, 6, 7, 8, 9];
	sShort		: STRING(10) := 'XAF';

	(* conversion buffer *)
	field1 : ARRAY[0..50 ] OF BYTE;
	field2 : ARRAY[0..50 ] OF BYTE;
	field3 : ARRAY[0..50 ] OF BYTE;
	field4 : ARRAY[0..50 ] OF BYTE;
	field5 : ARRAY[0..50 ] OF BYTE;
	field6 : ARRAY[0..50 ] OF BYTE;

	cbField1 : UDINT;
	cbField2 : UDINT;
	cbField3 : UDINT;
	cbField4 : UDINT;
	cbField5 : UDINT;
	cbField6 : UDINT;

	cbVar1 : UDINT;
	cbVar2 : UDINT;
	cbVar3 : UDINT;
	cbVar4 : UDINT;
	cbVar5 : UDINT;
	cbVar6 : UDINT;

END_VAR

cbField1 := ARG_TO_CSVFIELD( F_BOOL( bOperating ), TRUE, ADR( field1 ), SIZEOF( field1 ) );
cbField2 := ARG_TO_CSVFIELD( F_LREAL( fAxPos ), TRUE, ADR( field2 ), SIZEOF( field2 ) );
cbField3 := ARG_TO_CSVFIELD( F_UDINT( nCounter ), TRUE, ADR( field3 ), SIZEOF( field3 ) );
cbField4 := ARG_TO_CSVFIELD( F_STRING( sName ), TRUE, ADR( field4 ), SIZEOF( field4 ) );
cbField5 := ARG_TO_CSVFIELD( F_BIGTYPE( ADR( binData ), SIZEOF( binData ) ), TRUE, ADR( field5 ), SIZEOF( field5 ) );
cbField6 := ARG_TO_CSVFIELD( F_BIGTYPE( ADR( sShort ), INT_TO_DWORD( LEN( sShort ) ) ), TRUE, ADR( field6 ), SIZEOF( field6 ) );

cbVar1 := CSVFIELD_TO_ARG( ADR( field1 ), cbField1, TRUE, F_BOOL( bOperating ) );
cbVar2 := CSVFIELD_TO_ARG( ADR( field2 ), cbField2, TRUE, F_LREAL( fAxPos ) );
cbVar3 := CSVFIELD_TO_ARG( ADR( field3 ), cbField3, TRUE, F_UDINT( nCounter ) );
cbVar4 := CSVFIELD_TO_ARG( ADR( field4 ), cbField4, TRUE, F_STRING( sName ) );
cbVar5 := CSVFIELD_TO_ARG( ADR( field5 ), cbField5, TRUE, F_BIGTYPE( ADR( binData ), SIZEOF( binData ) ) );
cbVar6 := CSVFIELD_TO_ARG( ADR( field6 ), cbField6, TRUE, F_BIGTYPE( ADR( sShort ), INT_TO_DWORD( LEN( sShort ) ) ) );

END_PROGRAM

// ---- POUs/P_StringToConvExample.TcPOU
PROGRAM P_StringToConvExample
VAR
	s1	: STRING;
	s2	: STRING;
END_VAR

s1 := STRING_TO_CSVFIELD( 'Module_"ALFA_$05"_6', TRUE  );
s2 := STRING_TO_CSVFIELD( 'Module_50', FALSE );

s1 := CSVFIELD_TO_STRING( '"ab_$04_$05_cd-""ALFA""_5"', TRUE  );
s2 := CSVFIELD_TO_STRING( 'Module_50', FALSE );

END_PROGRAM

// ---- POUs/FunctionBlock/FB_AI_STATUS_Check.TcPOU
FUNCTION_BLOCK FB_AI_STATUS_Check
VAR_INPUT
	bEnable: BOOL;
	dwStatus: DWORD;
END_VAR
VAR_OUTPUT
	underrange: BOOL; 
	overrange: BOOL; 
	error: BOOL; 
END_VAR

IF bEnable THEN	
	underrange := GETBIT32(inVal32 := dwStatus, bitNo := 0);
	overrange := GETBIT32(inVal32 := dwStatus, bitNo := 1);
	error := GETBIT32(inVal32 := dwStatus, bitNo := 6);
END_IF

END_FUNCTION_BLOCK

// ---- POUs/FunctionBlock/FB_AVG10.TcPOU
FUNCTION_BLOCK FB_AVG10
VAR_INPUT
	fValue: REAL;
END_VAR
VAR_OUTPUT
	AVG: REAL := 0;
END_VAR
VAR
	Datas: ARRAY [0..9] OF REAL;
	Total: REAL := 0;	
    i: INT := 0;
	j: INT := 0;
END_VAR


IF i = 9 THEN
	//First In -> First Out
	FOR j := 1 TO 9 DO
		Datas[j-1] := Datas[j];
	END_FOR 
	Datas[9] := fValue;
ELSE
	Datas[i] := fValue;
	i := i + 1;
END_IF

Total := 0;
FOR j := 0 TO 9 DO
	Total := Total + Datas[j];
END_FOR 

AVG := Total / 10;

END_FUNCTION_BLOCK

// ---- POUs/FunctionBlock/FB_DeviationCheck.TcPOU
FUNCTION_BLOCK FB_DeviationCheck
VAR_INPUT
	bReset: BOOL;
	bEn_Alarm: BOOL;
	bEn_Warning: BOOL;
	fDeviPV: REAL;
	wAlarmDevi: WORD;
	dwAlarmCheckMilisec: DWORD;
	wWarningDevi: WORD;
	dwWarningCheckMilisec: DWORD;	
END_VAR
VAR_OUTPUT
	isAlarm : BOOL;
	isWarning : BOOL;
END_VAR
VAR
	T1 : TON;
	T2 : TON;
	wAlarmDev_Old : WORD;
	wWarnDev_Old : WORD;
	fAlarmDev : REAL;
	fWarnDev : REAL;
END_VAR

//Alarm Check
IF wAlarmDevi <> wAlarmDev_Old THEN
	wAlarmDev_Old := wAlarmDevi;
	fAlarmDev := WORD_TO_REAL(wAlarmDev_Old);
END_IF

T1();
T1.PT := DWORD_TO_TIME(dwAlarmCheckMilisec);
T1.IN := bEn_Alarm AND ABS(fDeviPV) > fAlarmDev AND isAlarm = FALSE ;
IF T1.Q THEN
	isAlarm := TRUE;
END_IF;


//Warning Check
IF wWarningDevi <> wWarnDev_Old THEN
	wWarnDev_Old := wWarningDevi;
	fWarnDev := WORD_TO_REAL(wWarnDev_Old);
END_IF

T2();
T2.PT := DWORD_TO_TIME(dwWarningCheckMilisec);
T2.IN := bEn_Warning AND ABS(fDeviPV) > fWarnDev AND isWarning = FALSE ;
IF T2.Q THEN
	isWarning := TRUE;
END_IF;

IF bReset THEN
	isAlarm := FALSE;	
	isWarning := FALSE;
END_IF

END_FUNCTION_BLOCK

// ---- POUs/FunctionBlock/FB_NoiseCheck.TcPOU
FUNCTION_BLOCK FB_NoiseCheck
VAR
	T1: TON;  (*타이머 *)
END_VAR
VAR_INPUT
	bEnable: BOOL;
	bReset: BOOL;
	bDI: BOOL;(*디지털 시그널*)
	wCheckMiliSec: WORD;(*딜레이 타임 millisecond*)
END_VAR
VAR_OUTPUT
	noNoise: BOOL; 
END_VAR

T1();
T1.PT := WORD_TO_TIME(wCheckMiliSec);
T1.IN := bEnable AND  bDI  AND noNoise = FALSE ;
IF T1.Q THEN
	noNoise := TRUE;
END_IF;

IF bReset THEN
	noNoise := FALSE;	
END_IF

END_FUNCTION_BLOCK

// ---- POUs/FunctionBlock/FB_PID.TcPOU
FUNCTION_BLOCK FB_PID
VAR_INPUT
	bRun: BOOL := FALSE;
	Kp: REAL;
	Ki: REAL;
	Kd: REAL;
	DeltaT: REAL;
    Pv: REAL;
	Sv: REAL;
END_VAR
VAR_OUTPUT
	control : REAL;
    prev_control : REAL;
	CtrlPercent : REAL;
    powerOn : BOOL;
END_VAR
VAR
	err : REAL;
	prev_err : REAL;
	I_err :	REAL;
	D_err : REAL;
	Kp_term : REAL;
	Ki_term : REAL;
	Kd_term : REAL;
END_VAR

IF bRun THEN
	err:= Sv - Pv; 	(* 오차 = 목표치-현재값*)
	Kp_term:= Kp *err;	(* P항 = Kp*오차  *)

	I_err := I_err + err * DeltaT; (* 오차적분 += 오차 * dt  *)
	Ki_term := Ki * I_err;	(*i항 = Ki * 오차적분*)

	D_err := (err-prev_err) / DeltaT; (*오차미분 = (현재오차-이전오차)/dt*)
	Kd_term := Kd * D_err; (*d항 =  Kd*오차미분*)

	prev_err := err; (*현재 오차를 이전 오차로*)
	control := Kp_term + Ki_term + Kd_term;(* 제어량 = p항 + i항 + d항*)

	powerOn :=   prev_control < control;
	CtrlPercent := (control - prev_control) / 100;
	prev_control := control;
ELSE
	powerOn := FALSE;
	CtrlPercent := prev_control := control := Kp_term := Ki_term := Kd_term := 0;
END_IF;

END_FUNCTION_BLOCK

// ---- POUs/FunctionBlock/FB_Ramp2.TcPOU
FUNCTION_BLOCK FB_Ramp2
VAR_INPUT
	bPause: BOOL;
	bReStart: BOOL;
	bStop: BOOL;
	tTimeUnit: TIME;
	fSV: REAL;	
	fSV_Step: REAL;
END_VAR
VAR_OUTPUT
	fyOut: REAL;
END_VAR
VAR_IN_OUT	
END_VAR
VAR
	T1: TON;
	fSV_Old: REAL;
	fSV_Step_Old: REAL;
	fSV_Inc: REAL;
	isPlus: BOOL;
	bT1_Rst: BOOL;
	bT1_On: BOOL;
END_VAR

T1(IN:=bT1_On, PT:=tTimeUnit);

//Check Input Value changed
IF fSV <> fSV_Old OR fSV_Step <> fSV_Step_Old THEN
	IF fSV_Step	<= 0 THEN 
		fSV_Step := 1; 
	END_IF	
    isPlus := fSV > fyOut;// Check Inc OR Dec
	fSV_Inc := (fyOut - fSV) / fSV_Step; //Calc Inc Value
    bT1_Rst := T1.ET <> T#0MS AND T1.Q = 0; //T1 Reset
END_IF

fSV_Old := fSV;
fSV_Step_Old := fSV_Step;

//T1 En Condition
bT1_On := bT1_Rst = 0 AND fSV <> fyOut;

IF bT1_Rst THEN
	bT1_Rst := 0;
ELSE//Ramping
	IF T1.Q THEN
		bT1_On := 0;//T1 Init
		IF bPause = 0 THEN
			fyOut := fyOut - fSV_Inc;
		END_IF
		
		IF isPlus = 0 AND fyOut < fSV THEN fyOut := fSV; END_IF
		IF isPlus = 1 AND fyOut > fSV THEN fyOut := fSV; END_IF
	END_IF
END_IF

IF fSV_Step = 1 THEN
	fyOut := fSV;
END_IF

IF bStop THEN
	fSV_Step := 1;
	fSV := fyOut;
END_IF

END_FUNCTION_BLOCK

// ---- POUs/FunctionBlock/FB_RampControl.TcPOU
FUNCTION_BLOCK FB_RampControl
VAR_INPUT
	bPause: BOOL;
	bReStart: BOOL;
	bStop: BOOL;
END_VAR
VAR_OUTPUT
	fyValue: REAL;
END_VAR
VAR_IN_OUT
	fSetValue: REAL;
	fSetRamp: REAL;
END_VAR
VAR
	Timer: TON;
	Step: INT;
	fSetValue_Copy: REAL;
	fSetRamp_Copy: REAL;
	fyValue_Copy: REAL;
	fRamp_Inc: REAL;
	fPause_SetValue_Copy: REAL;
	fPause_Ramp_Copy: REAL;
	isPaused: BOOL;
END_VAR

Timer();

(*사용자가 bPause버튼을 누르면 Ramp 멈추고 현재 값으로 유지*)
IF bPause = TRUE THEN
	IF isPaused = FALSE THEN
		fPause_Ramp_Copy :=	ABS( fSetRamp_Copy - fRamp_Inc);
		fPause_SetValue_Copy :=	fSetValue_Copy;
		fSetRamp := 0;
		fSetValue := fyValue;
		isPaused := TRUE;
	END_IF;
END_IF;

(*사용자가 bStop버튼을 누르면 Ramp 멈추고 현재 값으로 유지*)
IF bStop = TRUE THEN
	fSetRamp :=	0;
	fSetValue := fyValue;
END_IF;

(*bReStart 버튼을 누르면 재시작됨 *)
IF bReStart = TRUE THEN
	IF isPaused = TRUE THEN(*Puase 버튼이 정상적으로 눌린 경우만 *)
		fSetValue := fPause_SetValue_Copy;
		fSetRamp :=	fPause_Ramp_Copy;
		isPaused :=	FALSE;
		bReStart := FALSE;
		bPause := FALSE;
	END_IF;
END_IF;

//Ramp Process
CASE Step OF
	0:(*Input Change?*)
		IF	fSetValue_Copy	<>	fSetValue	THEN
			Step := 20;
		ELSE
			Step := 10;
		END_IF;

	10:(*Ramp Change?*)
		IF	fSetRamp_Copy <> fSetRamp		THEN
			Step := 20;
		ELSE
			Step := 0;
		END_IF;

	20:(*Input buf 저장*)
		fSetValue_Copy := fSetValue	;
		fSetRamp_Copy := fSetRamp;
		fyValue_Copy := fyValue;
		Step := 30;

	30: //Ramp Value Check
		IF fSetRamp	= 0	THEN
			fyValue := fSetValue_Copy;
			Step :=	0;
		ELSE
			Step :=	40;
		END_IF;

	40: //Ramp Variable Init
		fRamp_Inc := 0;
		Step :=	50;
		Timer.PT :=	T#1000MS;
		Timer.IN := FALSE;
		isPaused := FALSE;

	50:(*Timer*)
		Timer.IN := TRUE;

		IF Timer.Q = TRUE THEN(* Timer 1초가 되면 진행 *)
			Timer.IN := FALSE;
			fRamp_Inc := fRamp_Inc + 1;   (*Ramp 1초 증가  시킴*)
			fyValue	:=	fyValue + ((fSetValue_Copy   - fyValue_Copy ) / fSetRamp_Copy);  (*1초에 한번씩 output 증가 시킴*)

			IF fyValue <=0 THEN(*계산후 output 이 0 이하면 0으로 처리함*)
				fyValue := 0;
			END_IF;

			(*Ramp 종료 check*)
			IF fRamp_Inc >= fSetRamp THEN
				Step := 0;
			ELSE(*Ramp 변경??*)
				IF fSetRamp_Copy <> fSetRamp THEN
						(**???????????????????????????????????????????????????*)
					IF	fSetRamp <= 0 THEN
						Step := 0;
					ELSE
						fSetValue_Copy := fSetValue;
						fSetRamp_Copy := fSetRamp;
						fyValue_Copy := fyValue;
						Step := 40;
					END_IF;
				ELSE
					IF fSetValue_Copy <> fSetValue THEN(*Input 변경??*)
					fSetValue_Copy := fSetValue;
					fyValue_Copy := fyValue;
						IF fSetRamp	= 0 THEN
							Step := 0;
						ELSE
							Step := 40;
						END_IF;
					ELSE(*ramp Input 둘다 변경 없으면 Inc만 증가*)
						Step := 50;
					END_IF;
				END_IF;
			END_IF;
		END_IF;
END_CASE

END_FUNCTION_BLOCK

// ---- POUs/FunctionBlock/FB_Ramp_0.TcPOU
FUNCTION_BLOCK FB_Ramp_0
VAR_INPUT
	p_EN: BOOL;
	bRcpMode: BOOL;
	bPause: BOOL;
	bReStart: BOOL;
	bStop: BOOL;
	tTimeUnit: TIME;
	fSV: REAL;	
	fSV_Step: REAL;
END_VAR
VAR_OUTPUT
	fyOut : REAL;
END_VAR
VAR_IN_OUT	
END_VAR
VAR
	T1 : TON;
	fSV_Old : REAL;
	fSV_Step_Old  : REAL;
	fSV_Inc	   : REAL;
	isPlus : BOOL;
	bT1_Rst : BOOL;
	bT1_On : BOOL;
END_VAR

T1(IN:=bT1_On, PT:=tTimeUnit);

//Check Input Value changed
IF fSV <> fSV_Old OR fSV_Step <> fSV_Step_Old THEN
	IF fSV_Step	<= 0 THEN fSV_Step := 1; END_IF	// Limit Check
    isPlus := fSV > fyOut;// Check Inc OR Dec
	fSV_Inc := (fyOut - fSV) / fSV_Step; //Calc Inc Value
    bT1_Rst := T1.ET <> T#0MS AND T1.Q = 0; //T1 Reset
END_IF

fSV_Old := fSV;
fSV_Step_Old := fSV_Step;

//T1 En Condition
bT1_On := bT1_Rst = 0 AND fSV <> fyOut;

IF bRcpMode = Off THEN	
	IF bT1_Rst THEN
		bT1_Rst := 0;
	ELSE//Ramping
		IF T1.Q THEN
			bT1_On := 0;//T1 Init
			IF bPause = 0 THEN fyOut := fyOut - fSV_Inc; END_IF				
			IF isPlus = 0 AND fyOut < fSV THEN fyOut := fSV; END_IF
			IF isPlus = 1 AND fyOut > fSV THEN fyOut := fSV; END_IF
		END_IF
	END_IF
ELSE
	IF p_EN THEN		
		IF bPause = 0 THEN fyOut := fyOut - fSV_Inc; END_IF			
		IF isPlus = 0 AND fyOut < fSV THEN fyOut := fSV; END_IF
		IF isPlus = 1 AND fyOut > fSV THEN fyOut := fSV; END_IF
	END_IF	
END_IF


IF fSV_Step = 1 THEN
	fyOut := fSV;
END_IF

IF bStop THEN
	fSV_Step := 1;
	fSV := fyOut;
END_IF

END_FUNCTION_BLOCK

// ---- POUs/FunctionBlock/FB_RcpRamp.TcPOU
FUNCTION_BLOCK FB_RcpRamp
VAR_INPUT
	pEN: BOOL;
	bPause: BOOL;	
	bStop: BOOL;
	fSV: REAL;	
	fSV_Step: REAL;
END_VAR
VAR_OUTPUT
	fyOut: REAL;
END_VAR
VAR_IN_OUT	
END_VAR
VAR
	fSV_Old: REAL;
	fSV_Step_Old: REAL;
	fSV_Inc: REAL;
	isPlus: BOOL;
END_VAR


//Check Input Value changed
IF fSV <> fSV_Old OR fSV_Step <> fSV_Step_Old THEN
	IF fSV_Step	<= 0 THEN 
		fSV_Step := 1; 
	END_IF	
    isPlus := fSV > fyOut;// Check Inc OR Dec
	fSV_Inc := (fyOut - fSV) / fSV_Step; //Calc Inc Value   
END_IF

fSV_Old := fSV;
fSV_Step_Old := fSV_Step;

//Ramping
IF pEN THEN
	IF bPause = 0 THEN
		fyOut := fyOut - fSV_Inc;
	END_IF
		
	IF isPlus = 0 AND fyOut < fSV THEN fyOut := fSV; END_IF
	IF isPlus = 1 AND fyOut > fSV THEN fyOut := fSV; END_IF
END_IF


IF fSV_Step = 1 THEN
	fyOut := fSV;
END_IF

IF bStop THEN
	fSV_Step := 1;
	fSV := fyOut;
END_IF


//T1(IN:=bT1_On, PT:=tTimeUnit);

END_FUNCTION_BLOCK

// ---- POUs/Function/F_ET2Sec.TcPOU
FUNCTION F_ET2Sec : REAL
VAR_INPUT
	IN: TIME;
	SecScale: REAL;
END_VAR
VAR
	r1: REAL;
END_VAR


r1:= TIME_TO_REAL(IN);
IF r1 > 0 THEN
	F_ET2Sec := r1 / SecScale;
ELSE
	F_ET2Sec := 0;	
END_IF

END_FUNCTION

// ---- POUs/Function/F_Int2Real.TcPOU
FUNCTION F_Int2Real : REAL
VAR_INPUT
	nIn: INT;
	nDecimal: INT;
END_VAR
VAR
	rVal: REAL;
END_VAR

rVal:= INT_TO_REAL(nIn);	
CASE nDecimal OF
	1:  
		rVal := rVal / 10;
	2:     
		rVal := rVal / 100;
	3:
		rVal := rVal / 1000;    
END_CASE;
F_Int2Real := rVal;

END_FUNCTION

// ---- POUs/Function/F_LH_PV.TcPOU
FUNCTION F_LH_PV : REAL
VAR_INPUT
	hexPV: STRING;
	nDecimal: INT := 0;
END_VAR
VAR
	data: ARRAY[0..1] OF BYTE;
	b1: BYTE;
	cbData: UDINT;
	ptPV: POINTER TO INT;
	iPV: INT;
	i: INT;
	r1: REAL;
END_VAR


cbData := HEXSTR_TO_DATA(hexPV, ADR(data), SIZEOF(data));
		
//Swap
b1 := data[0];
data[0] := data[1];
data[1] := b1;
		
ptPV := ADR(data);
iPV := ptPV^;
r1 := INT_TO_REAL(iPV);

//Decimal
FOR i := 0 TO nDecimal - 1 BY 1 DO
	r1 := r1 / 10;
END_FOR

F_LH_PV := r1;

END_FUNCTION

// ---- POUs/Function/F_LH_SV.TcPOU
FUNCTION F_LH_SV : string
VAR_INPUT
	SV: REAL;
	nDecimal: INT := 0;
END_VAR
VAR
	iPV: INT;
	wPV: WORD;
	i: INT;
	r1: REAL;
END_VAR


r1 := SV;

//Decimal
FOR i := 0 TO nDecimal - 1 BY 1 DO
	r1 := r1 * 10;
END_FOR

iPV := REAL_TO_INT(r1);
wPV := INT_TO_WORD(iPV);

F_LH_SV := WORD_TO_HEXSTR(in:= wPV, iPrecision:= 4, bLoCase:= FALSE);

END_FUNCTION

// ---- POUs/Function/F_OPSTATE.TcPOU
FUNCTION F_OPSTATE : BOOL
VAR_INPUT
	uStateIn: UINT;
END_VAR
VAR
END_VAR

F_OPSTATE := GETBIT32(inVal32 := uStateIn, bitNo := 3);

END_FUNCTION

// ---- POUs/Function/F_TB_PV2REAL.TcPOU
FUNCTION F_TB_PV2REAL : REAL
VAR_INPUT
	PvStr: STRING;
END_VAR
VAR
	iPV: LINT;
	r1: REAL;
END_VAR

// SMC HEBC002-WA10
// sv >= 0 -> '00010'
// sv < 0 -> '-0010'
iPV := STRING_TO_LINT(PvStr);
r1 := LINT_TO_REAL(iPV);
F_TB_PV2REAL := r1 / 10;

END_FUNCTION

// ---- POUs/Function/F_TB_Rx_BCC.TcPOU
FUNCTION F_TB_Rx_BCC : BOOL
VAR_INPUT
	rxStr: STRING;
END_VAR
VAR
	i, len1, len2: INT;
	bArr: ARRAY[0..255] OF BYTE;
	b1: BYTE;
END_VAR

// SMC HEBC002-WA10
len1 := LEN(STR:=rxStr);
len2 := len1;
len1 := len1 - 1;
bArr := MAXSTRING_TO_BYTEARR(rxStr);
FOR i := 0 TO len1 DO
	b1 := b1 XOR bArr[i];
END_FOR
F_TB_Rx_BCC := b1 = bArr[len2];

END_FUNCTION

// ---- POUs/Function/F_TB_SV2STR.TcPOU
FUNCTION F_TB_SV2STR : STRING
VAR_INPUT
	SV: REAL;
END_VAR
VAR
	r1: REAL;
	iSV: LINT;
	str: STRING;
END_VAR

// SMC HEBC002-WA10
// sv >= 0 -> '00010'
// sv < 0 -> '-0010'
r1 := SV * 10;
iSV := REAL_TO_LINT(r1);
IF iSV >= 0 THEN
	str := LINT_TO_DECSTR(in:=iSV, iPrecision:=5);
ELSE
	str := CONCAT('', LINT_TO_DECSTR(in:=iSV, iPrecision:=4));	//CONCAT('-', LINT_TO_DECSTR(in:=iSV, iPrecision:=4));	
END_IF
F_TB_SV2STR := str;

END_FUNCTION

// ---- POUs/Function/F_TB_Tx_BCC.TcPOU
FUNCTION F_TB_Tx_BCC : STRING
VAR_INPUT
	txStr: STRING;
END_VAR
VAR
	i, len1: INT;
	bArr: ARRAY[0..255] OF BYTE;
	b1: BYTE;
END_VAR

// SMC HEBC002-WA10
len1 := LEN(STR:=txStr);
len1 := len1 - 1;
bArr := MAXSTRING_TO_BYTEARR(txStr);
FOR i := 0 TO len1 DO
	b1 := b1 XOR bArr[i];
END_FOR
F_TB_Tx_BCC := F_toCHR(b1);

END_FUNCTION

// ---- POUs/MR_PRG/P00_Main.TcPOU
PROGRAM P00_Main
VAR
	netID: T_AmsNetID;// := '10.10.10.10.1.1';
	fbNetId: FB_GetLocalAmsNetId;
	fbRestart: TC_Restart;
	idx: INT;
	bOpState: BOOL;
    bTCAT_Net_err: BOOL;	
END_VAR

IF cm_TCAT_restart THEN		
	fbNetId(bExecute := cm_TCAT_restart, tTimeOut := T#1S);	
	IF fbNetId.bBusy = 0 THEN
		cm_TCAT_restart := 0;
		netID := fbNetId.AddrString;
		fbRestart(NETID := netID, RESTART := 1);
	END_IF	
END_IF


bOpState := 1;
FOR idx := 0 TO 1 DO
	IF N_COUPLER_STATES[idx] <> 0 THEN
		bOpState := 0;
		EXIT;
	END_IF
END_FOR
is_TCAT_OpState := bOpState;

bTCAT_Net_err := 0;
FOR idx := 0 TO 6 DO
	IF N_NET_STATES[idx] <> 0 THEN
		bTCAT_Net_err := 1;
		EXIT;
	END_IF
END_FOR   
is_TCAT_Net_err := bTCAT_Net_err;

IF is_TCAT_OpState THEN		
	P00_OP();
	//Init
	P01_Init_N_Retain();
    P02_Init_MC();
    	
	//Communication
	P02_P2P();
	
	//Input
	//REF_P02_KL1501();
	P11_Rx_TV();
	P12_Rx_IH();
	P13_DI_N_Check();
	P15_AI();
	//Check
	
	ACT_Status_Check();
	
	//Process
	P21_AL_WN();
	IF ing_FC = 0 AND is_RCP_runable AND cm_RCP_start THEN
		s_EN_EXE_RCP := NOT is_AL;		
	END_IF
		
	IF (di_SH_lo_limit AND di_VP_busy ) AND (cm_DOR_VAC OR di_DOR_VAC )THEN //di_PUMP_fail is B Contact
		s_EN_EXE_DOR_ATM := 0;
		s_EN_EXE_DOR_VAC := NOT is_AL;		
	END_IF
	IF s_EN_EXE_DOR_VAC AND cm_FC_stop THEN
		s_EN_EXE_DOR_VAC := 0;		
	END_IF
	
	IF EN_DOR_ATM AND (cm_DOR_ATM OR di_DOR_ATM) THEN
		s_EN_EXE_DOR_VAC := 0;
		s_EN_EXE_DOR_ATM := NOT is_AL;		
	END_IF	
	IF s_EN_EXE_DOR_ATM AND cm_FC_stop THEN
		s_EN_EXE_DOR_ATM := 0;		
	END_IF	
	
	IF ing_FC = 0 AND cm_ROT_caliStart THEN
		s_EN_EXE_ROT_CALI := NOT is_AL;		
	END_IF	
	
	IF s_EN_EXE_ROT_CALI AND cm_FC_stop THEN
		s_EN_EXE_ROT_CALI := 0;		
	END_IF	

	P22_RCP_Ctrl();	
	P24_Rot_Calibration();
	P25_US_Ctrl();
	
	//Etc
	P31_BypassV();
	P41_DOR_VAC();
	P41_DOR_Vac_Check();
	P42_DOR_ATM();
	P43_SH_UpDw();
	P49_MO_SRC();
		
	//Output	
	P62_Tx_TV();
	P63_Tx_IH();
	P53_DO_VV();
	P54_DO_ETC();
	P61_AO();
		
	cm_FC_stop := 0;		
	cm_RCP_start := 0;
	cm_DOR_VAC := 0;
	cm_DOR_ATM := 0;	
	cm_ROT_caliStart := 0;
		
END_IF

ing_FC := s_EN_EXE_RCP OR s_EN_EXE_DOR_VAC OR s_EN_EXE_DOR_ATM OR s_EN_EXE_ROT_CALI;

IF ing_FC THEN
	IF s_EN_EXE_RCP THEN pv_FC_ID := 1; END_IF
	IF s_EN_EXE_DOR_VAC THEN pv_FC_ID := 2; END_IF
	IF s_EN_EXE_DOR_ATM THEN pv_FC_ID := 3; END_IF
	IF s_EN_EXE_ROT_CALI THEN pv_FC_ID := 4; END_IF
ELSE
	pv_FC_ID := 0;
END_IF

ACTION ACT_Status_Check:
is_RCP_runable := is_TCAT_Net_err = 0 AND is_AL = 0 AND is_RCP_loaded 
				  AND di_VP_busy AND is_DOR_VAC_ok;// AND di_IH_ready;

IF e_d_AUTO_IH_on AND sv_IH >= 1 AND is_AL = 0 THEN cm_IH := 1; END_IF;
IF sv_IH < 1 OR en_SH_UpDw THEN cm_IH := 0; END_IF;
IF e_d_AUTO_ROT_on AND pv_ROT < 1 AND sv_ROT >= 1 AND is_AL = 0 THEN cm_ROT := 1; END_IF;
IF s_EN_ROT_JOG = 0 AND s_EN_ROT_INCH = 0 AND cm_ROT AND sv_ROT < 1 THEN cm_ROT := 0; END_IF;
END_ACTION

END_PROGRAM

// ---- POUs/MR_PRG/P00_OP.TcPOU
PROGRAM P00_OP
VAR		
	N_OP_CMD AT%MB64:  ARRAY [0..35] OF BYTE;//op cmd 주소
	memSetResult: UDINT;	
	b_Test: BOOL;
END_VAR
VAR // added by the converter: edge detectors and wires of the graphical bodies
    _rt1, _rt2, _rt3, _rt4, _rt5, _rt6, _rt7, _rt8, _rt9, _rt10, _rt11, _rt12, _rt13, _rt14, _rt15, _rt16, _rt17, _rt18, _rt19, _rt20, _rt21, _rt22, _rt23, _rt24, _rt25, _rt26, _rt27, _rt28, _rt29, _rt30, _rt31, _rt32, _rt33, _rt34, _rt35, _rt36, _rt37, _rt38, _rt39, _rt40, _rt41, _rt42, _rt43, _rt44, _rt45, _rt46, _rt47, _rt48, _rt49, _rt50, _rt51, _rt52, _rt53, _rt54, _rt55, _rt56, _rt57, _rt58, _rt59, _rt60, _rt61, _rt62, _rt63, _rt64, _rt65, _rt66, _rt67, _rt68, _rt69, _rt70, _rt71, _rt72, _rt73, _rt74, _rt75, _rt76, _rt77, _rt78, _rt79, _rt80, _rt81, _rt82, _rt83, _rt84, _rt85, _rt86, _rt87, _rt88, _rt89, _rt90, _rt91, _rt92, _rt93, _rt94, _rt95, _rt96, _rt97, _rt98, _rt99, _rt100, _rt101, _rt102, _rt103, _rt104, _rt105, _rt106, _rt107, _rt108, _rt109, _rt110, _rt111, _rt112, _rt113, _rt114, _rt115, _rt116, _rt117, _rt118, _rt119, _rt120, _rt121, _rt122, _rt123, _rt124, _rt125, _rt126, _rt127, _rt128, _rt129, _rt130, _rt131, _rt132, _rt133, _rt134, _rt135, _rt136, _rt137, _rt138, _rt139, _rt140, _rt141, _rt142, _rt143, _rt144, _rt145, _rt146, _rt147, _rt148, _rt149, _rt150, _rt151, _rt152, _rt153, _rt154, _rt155, _rt156, _rt157, _rt158, _rt159, _rt160, _rt161, _rt162, _rt163, _rt164, _rt165, _rt166, _rt167, _rt168, _rt169, _rt170, _rt171, _rt172, _rt173, _rt174, _rt175, _rt176, _rt177, _rt178, _rt179, _rt180, _rt181, _rt182, _rt183, _rt184, _rt185, _rt186, _rt187, _rt188, _rt189, _rt190, _rt191, _rt192, _rt193, _rt194, _rt195, _rt196, _rt197, _rt198, _rt199, _rt200, _rt201, _rt202, _rt203, _rt204, _rt205, _rt206, _rt207, _rt208, _rt209, _rt210, _rt211, _rt212, _rt213, _rt214, _rt215, _rt216, _rt217, _rt218, _rt219, _rt220, _rt221, _rt222, _rt223, _rt224, _rt225, _rt226, _rt227, _rt228, _rt229, _rt230, _rt231, _rt232, _rt233, _rt234 : R_TRIG;
    _w1, _w2, _w3, _w4, _w5, _w6, _w7, _w8, _w9, _w10, _w11, _w12 : BOOL;
END_VAR

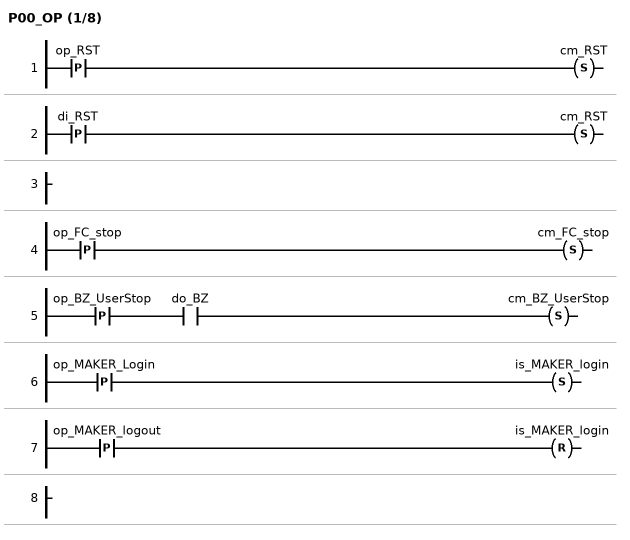
// NETWORK 1
_rt1(CLK := op_RST);
cm_RST S= _rt1.Q;

// NETWORK 2
_rt2(CLK := di_RST);
cm_RST S= _rt2.Q;

// NETWORK 3

// NETWORK 4
_rt3(CLK := op_FC_stop);
cm_FC_stop S= _rt3.Q;

// NETWORK 5
_rt4(CLK := op_BZ_UserStop);
cm_BZ_UserStop S= _rt4.Q AND do_BZ;

// NETWORK 6
_rt5(CLK := op_MAKER_Login);
is_MAKER_login S= _rt5.Q;

// NETWORK 7
_rt6(CLK := op_MAKER_logout);
is_MAKER_login R= _rt6.Q;

// NETWORK 8

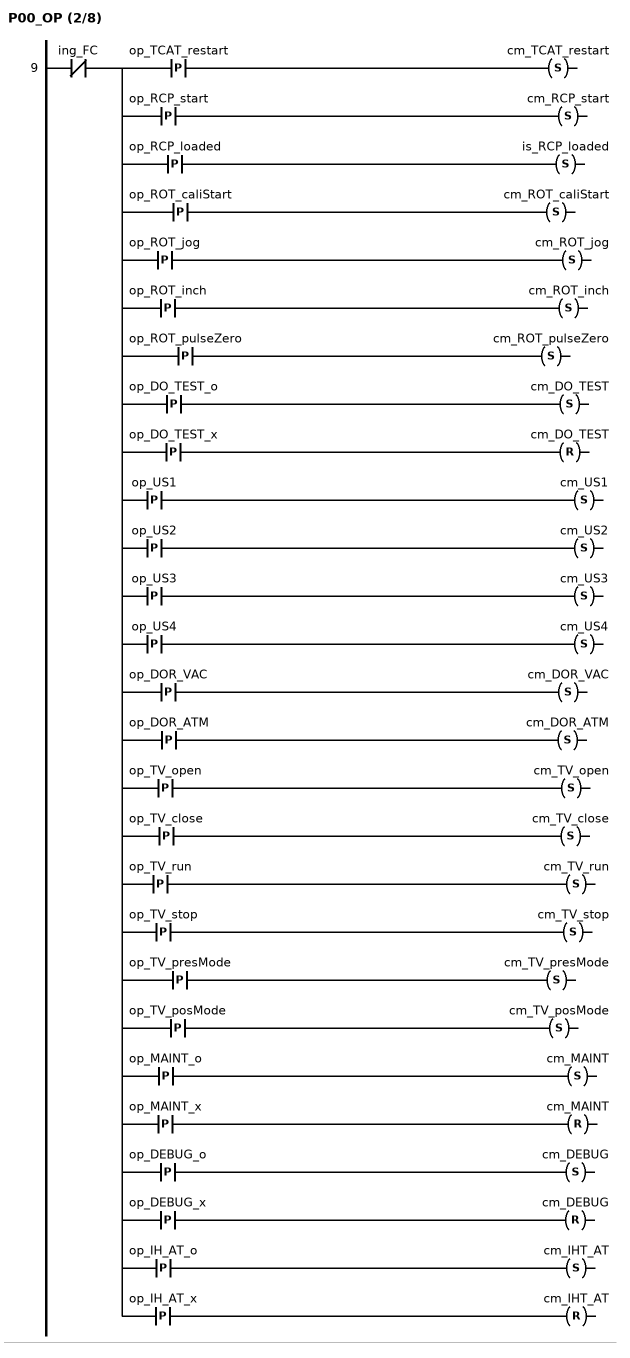
// NETWORK 9
_w1 := NOT ing_FC;
_rt7(CLK := op_TCAT_restart);
cm_TCAT_restart S= _w1 AND _rt7.Q;
_rt8(CLK := op_RCP_start);
cm_RCP_start S= _w1 AND _rt8.Q;
_rt9(CLK := op_RCP_loaded);
is_RCP_loaded S= _w1 AND _rt9.Q;
_rt10(CLK := op_ROT_caliStart);
cm_ROT_caliStart S= _w1 AND _rt10.Q;
_rt11(CLK := op_ROT_jog);
cm_ROT_jog S= _w1 AND _rt11.Q;
_rt12(CLK := op_ROT_inch);
cm_ROT_inch S= _w1 AND _rt12.Q;
_rt13(CLK := op_ROT_pulseZero);
cm_ROT_pulseZero S= _w1 AND _rt13.Q;
_rt14(CLK := op_DO_TEST_o);
cm_DO_TEST S= _w1 AND _rt14.Q;
_rt15(CLK := op_DO_TEST_x);
cm_DO_TEST R= _w1 AND _rt15.Q;
_rt16(CLK := op_US1);
cm_US1 S= _w1 AND _rt16.Q;
_rt17(CLK := op_US2);
cm_US2 S= _w1 AND _rt17.Q;
_rt18(CLK := op_US3);
cm_US3 S= _w1 AND _rt18.Q;
_rt19(CLK := op_US4);
cm_US4 S= _w1 AND _rt19.Q;
_rt20(CLK := op_DOR_VAC);
cm_DOR_VAC S= _w1 AND _rt20.Q;
_rt21(CLK := op_DOR_ATM);
cm_DOR_ATM S= _w1 AND _rt21.Q;
_rt22(CLK := op_TV_open);
cm_TV_open S= _w1 AND _rt22.Q;
_rt23(CLK := op_TV_close);
cm_TV_close S= _w1 AND _rt23.Q;
_rt24(CLK := op_TV_run);
cm_TV_run S= _w1 AND _rt24.Q;
_rt25(CLK := op_TV_stop);
cm_TV_stop S= _w1 AND _rt25.Q;
_rt26(CLK := op_TV_presMode);
cm_TV_presMode S= _w1 AND _rt26.Q;
_rt27(CLK := op_TV_posMode);
cm_TV_posMode S= _w1 AND _rt27.Q;
_rt28(CLK := op_MAINT_o);
cm_MAINT S= _w1 AND _rt28.Q;
_rt29(CLK := op_MAINT_x);
cm_MAINT R= _w1 AND _rt29.Q;
_rt30(CLK := op_DEBUG_o);
cm_DEBUG S= _w1 AND _rt30.Q;
_rt31(CLK := op_DEBUG_x);
cm_DEBUG R= _w1 AND _rt31.Q;
_rt32(CLK := op_IH_AT_o);
cm_IHT_AT S= _w1 AND _rt32.Q;
_rt33(CLK := op_IH_AT_x);
cm_IHT_AT R= _w1 AND _rt33.Q;

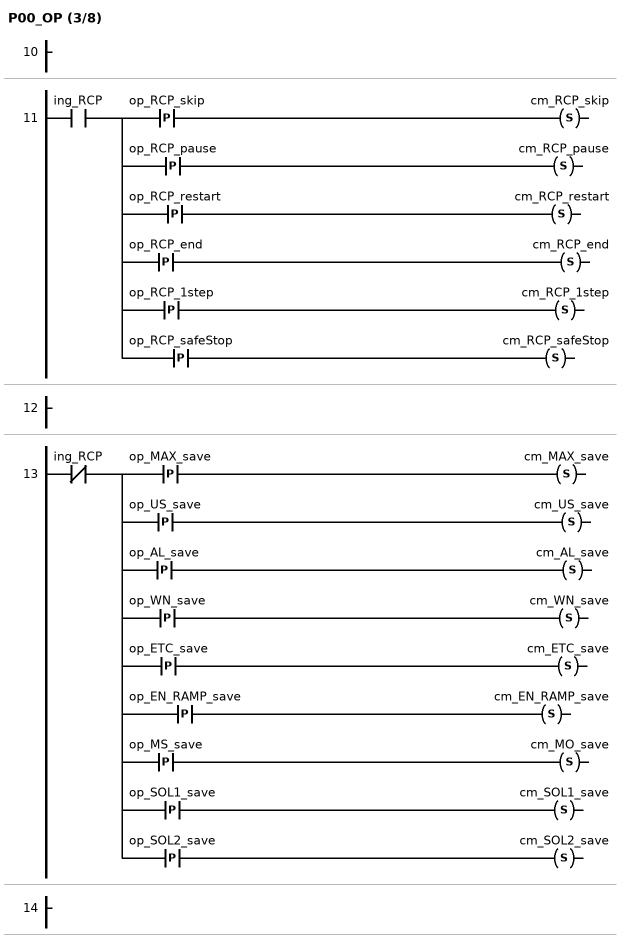
// NETWORK 10

// NETWORK 11
_rt34(CLK := op_RCP_skip);
cm_RCP_skip S= ing_RCP AND _rt34.Q;
_rt35(CLK := op_RCP_pause);
cm_RCP_pause S= ing_RCP AND _rt35.Q;
_rt36(CLK := op_RCP_restart);
cm_RCP_restart S= ing_RCP AND _rt36.Q;
_rt37(CLK := op_RCP_end);
cm_RCP_end S= ing_RCP AND _rt37.Q;
_rt38(CLK := op_RCP_1step);
cm_RCP_1step S= ing_RCP AND _rt38.Q;
_rt39(CLK := op_RCP_safeStop);
cm_RCP_safeStop S= ing_RCP AND _rt39.Q;

// NETWORK 12

// NETWORK 13
_w2 := NOT ing_RCP;
_rt40(CLK := op_MAX_save);
cm_MAX_save S= _w2 AND _rt40.Q;
_rt41(CLK := op_US_save);
cm_US_save S= _w2 AND _rt41.Q;
_rt42(CLK := op_AL_save);
cm_AL_save S= _w2 AND _rt42.Q;
_rt43(CLK := op_WN_save);
cm_WN_save S= _w2 AND _rt43.Q;
_rt44(CLK := op_ETC_save);
cm_ETC_save S= _w2 AND _rt44.Q;
_rt45(CLK := op_EN_RAMP_save);
cm_EN_RAMP_save S= _w2 AND _rt45.Q;
_rt46(CLK := op_MS_save);
cm_MO_save S= _w2 AND _rt46.Q;
_rt47(CLK := op_SOL1_save);
cm_SOL1_save S= _w2 AND _rt47.Q;
_rt48(CLK := op_SOL2_save);
cm_SOL2_save S= _w2 AND _rt48.Q;

// NETWORK 14

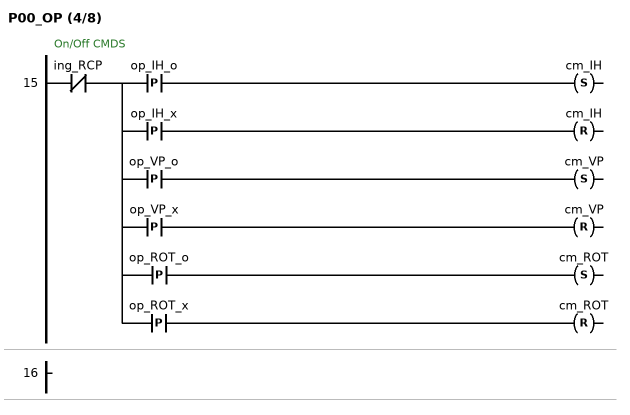
// NETWORK 15
// On/Off CMDS
_w3 := NOT ing_RCP;
_rt49(CLK := op_IH_o);
cm_IH S= _w3 AND _rt49.Q;
_rt50(CLK := op_IH_x);
cm_IH R= _w3 AND _rt50.Q;
_rt51(CLK := op_VP_o);
cm_VP S= _w3 AND _rt51.Q;
_rt52(CLK := op_VP_x);
cm_VP R= _w3 AND _rt52.Q;
_rt53(CLK := op_ROT_o);
cm_ROT S= _w3 AND _rt53.Q;
_rt54(CLK := op_ROT_x);
cm_ROT R= _w3 AND _rt54.Q;

// NETWORK 16

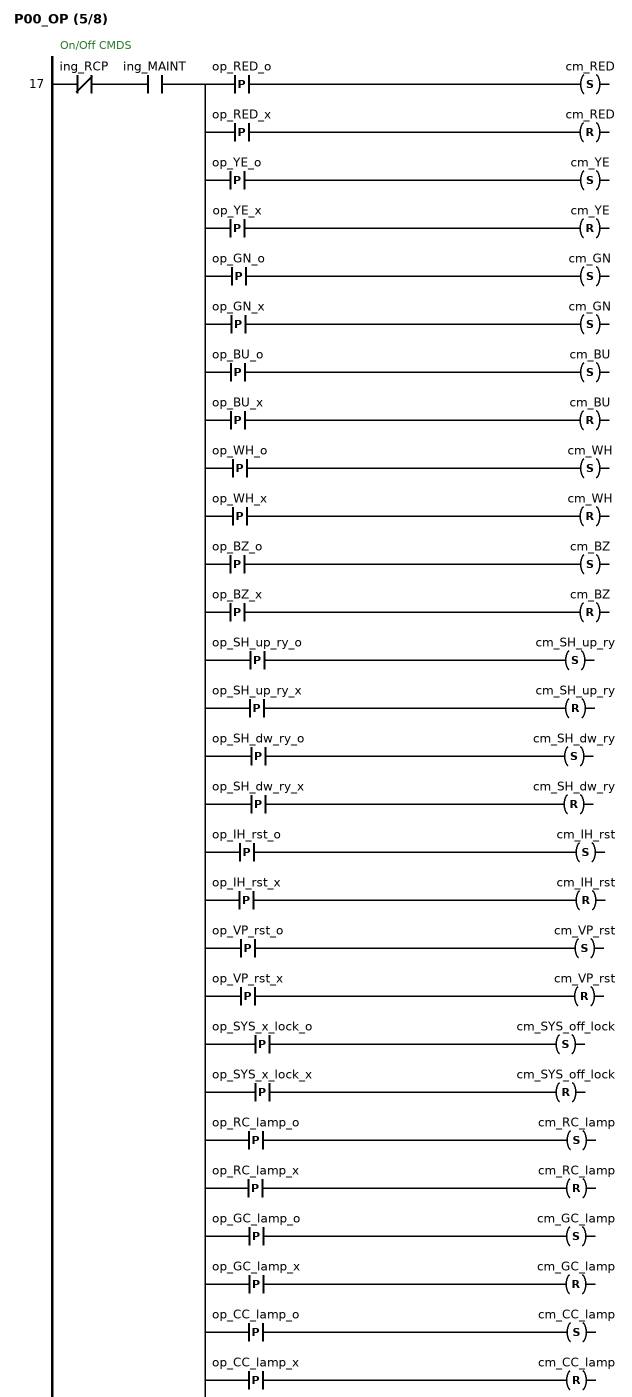
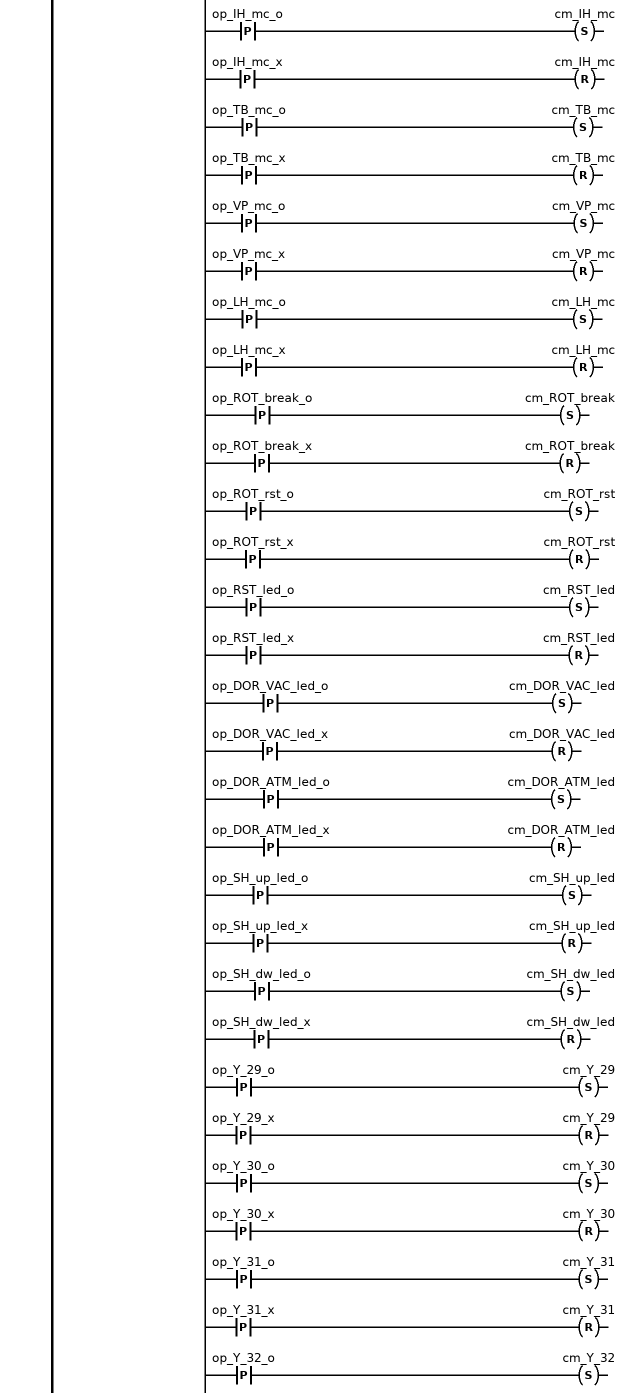
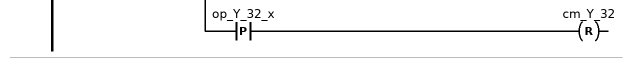
// NETWORK 17
// On/Off CMDS
_w4 := NOT ing_RCP AND ing_MAINT;
_rt55(CLK := op_RED_o);
cm_RED S= _w4 AND _rt55.Q;
_rt56(CLK := op_RED_x);
cm_RED R= _w4 AND _rt56.Q;
_rt57(CLK := op_YE_o);
cm_YE S= _w4 AND _rt57.Q;
_rt58(CLK := op_YE_x);
cm_YE R= _w4 AND _rt58.Q;
_rt59(CLK := op_GN_o);
cm_GN S= _w4 AND _rt59.Q;
_rt60(CLK := op_GN_x);
cm_GN S= _w4 AND _rt60.Q;
_rt61(CLK := op_BU_o);
cm_BU S= _w4 AND _rt61.Q;
_rt62(CLK := op_BU_x);
cm_BU R= _w4 AND _rt62.Q;
_rt63(CLK := op_WH_o);
cm_WH S= _w4 AND _rt63.Q;
_rt64(CLK := op_WH_x);
cm_WH R= _w4 AND _rt64.Q;
_rt65(CLK := op_BZ_o);
cm_BZ S= _w4 AND _rt65.Q;
_rt66(CLK := op_BZ_x);
cm_BZ R= _w4 AND _rt66.Q;
_rt67(CLK := op_SH_up_ry_o);
cm_SH_up_ry S= _w4 AND _rt67.Q;
_rt68(CLK := op_SH_up_ry_x);
cm_SH_up_ry R= _w4 AND _rt68.Q;
_rt69(CLK := op_SH_dw_ry_o);
cm_SH_dw_ry S= _w4 AND _rt69.Q;
_rt70(CLK := op_SH_dw_ry_x);
cm_SH_dw_ry R= _w4 AND _rt70.Q;
_rt71(CLK := op_IH_rst_o);
cm_IH_rst S= _w4 AND _rt71.Q;
_rt72(CLK := op_IH_rst_x);
cm_IH_rst R= _w4 AND _rt72.Q;
_rt73(CLK := op_VP_rst_o);
cm_VP_rst S= _w4 AND _rt73.Q;
_rt74(CLK := op_VP_rst_x);
cm_VP_rst R= _w4 AND _rt74.Q;
_rt75(CLK := op_SYS_x_lock_o);
cm_SYS_off_lock S= _w4 AND _rt75.Q;
_rt76(CLK := op_SYS_x_lock_x);
cm_SYS_off_lock R= _w4 AND _rt76.Q;
_rt77(CLK := op_RC_lamp_o);
cm_RC_lamp S= _w4 AND _rt77.Q;
_rt78(CLK := op_RC_lamp_x);
cm_RC_lamp R= _w4 AND _rt78.Q;
_rt79(CLK := op_GC_lamp_o);
cm_GC_lamp S= _w4 AND _rt79.Q;
_rt80(CLK := op_GC_lamp_x);
cm_GC_lamp R= _w4 AND _rt80.Q;
_rt81(CLK := op_CC_lamp_o);
cm_CC_lamp S= _w4 AND _rt81.Q;
_rt82(CLK := op_CC_lamp_x);
cm_CC_lamp R= _w4 AND _rt82.Q;
_rt83(CLK := op_IH_mc_o);
cm_IH_mc S= _w4 AND _rt83.Q;
_rt84(CLK := op_IH_mc_x);
cm_IH_mc R= _w4 AND _rt84.Q;
_rt85(CLK := op_TB_mc_o);
cm_TB_mc S= _w4 AND _rt85.Q;
_rt86(CLK := op_TB_mc_x);
cm_TB_mc R= _w4 AND _rt86.Q;
_rt87(CLK := op_VP_mc_o);
cm_VP_mc S= _w4 AND _rt87.Q;
_rt88(CLK := op_VP_mc_x);
cm_VP_mc R= _w4 AND _rt88.Q;
_rt89(CLK := op_LH_mc_o);
cm_LH_mc S= _w4 AND _rt89.Q;
_rt90(CLK := op_LH_mc_x);
cm_LH_mc R= _w4 AND _rt90.Q;
_rt91(CLK := op_ROT_break_o);
cm_ROT_break S= _w4 AND _rt91.Q;
_rt92(CLK := op_ROT_break_x);
cm_ROT_break R= _w4 AND _rt92.Q;
_rt93(CLK := op_ROT_rst_o);
cm_ROT_rst S= _w4 AND _rt93.Q;
_rt94(CLK := op_ROT_rst_x);
cm_ROT_rst R= _w4 AND _rt94.Q;
_rt95(CLK := op_RST_led_o);
cm_RST_led S= _w4 AND _rt95.Q;
_rt96(CLK := op_RST_led_x);
cm_RST_led R= _w4 AND _rt96.Q;
_rt97(CLK := op_DOR_VAC_led_o);
cm_DOR_VAC_led S= _w4 AND _rt97.Q;
_rt98(CLK := op_DOR_VAC_led_x);
cm_DOR_VAC_led R= _w4 AND _rt98.Q;
_rt99(CLK := op_DOR_ATM_led_o);
cm_DOR_ATM_led S= _w4 AND _rt99.Q;
_rt100(CLK := op_DOR_ATM_led_x);
cm_DOR_ATM_led R= _w4 AND _rt100.Q;
_rt101(CLK := op_SH_up_led_o);
cm_SH_up_led S= _w4 AND _rt101.Q;
_rt102(CLK := op_SH_up_led_x);
cm_SH_up_led R= _w4 AND _rt102.Q;
_rt103(CLK := op_SH_dw_led_o);
cm_SH_dw_led S= _w4 AND _rt103.Q;
_rt104(CLK := op_SH_dw_led_x);
cm_SH_dw_led R= _w4 AND _rt104.Q;
_rt105(CLK := op_Y_29_o);
cm_Y_29 S= _w4 AND _rt105.Q;
_rt106(CLK := op_Y_29_x);
cm_Y_29 R= _w4 AND _rt106.Q;
_rt107(CLK := op_Y_30_o);
cm_Y_30 S= _w4 AND _rt107.Q;
_rt108(CLK := op_Y_30_x);
cm_Y_30 R= _w4 AND _rt108.Q;
_rt109(CLK := op_Y_31_o);
cm_Y_31 S= _w4 AND _rt109.Q;
_rt110(CLK := op_Y_31_x);
cm_Y_31 R= _w4 AND _rt110.Q;
_rt111(CLK := op_Y_32_o);
cm_Y_32 S= _w4 AND _rt111.Q;
_rt112(CLK := op_Y_32_x);
cm_Y_32 R= _w4 AND _rt112.Q;

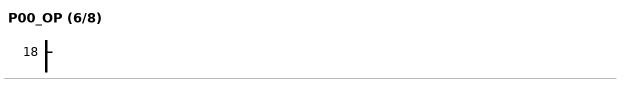
// NETWORK 18

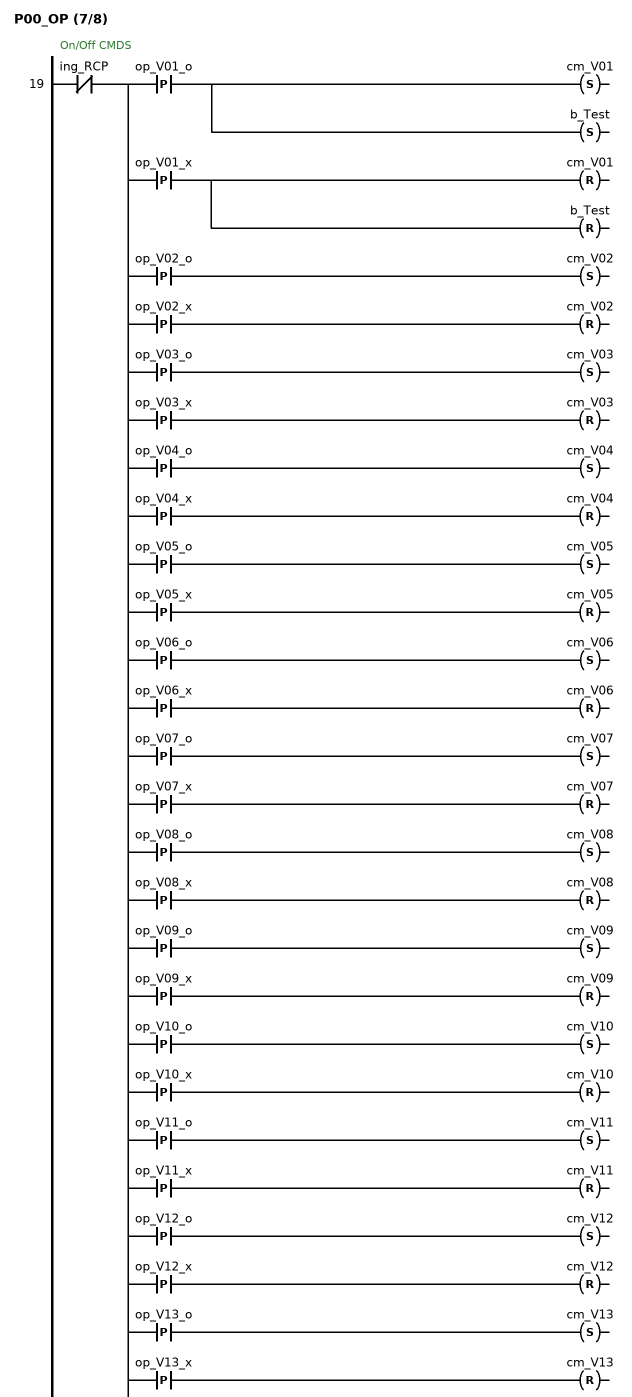
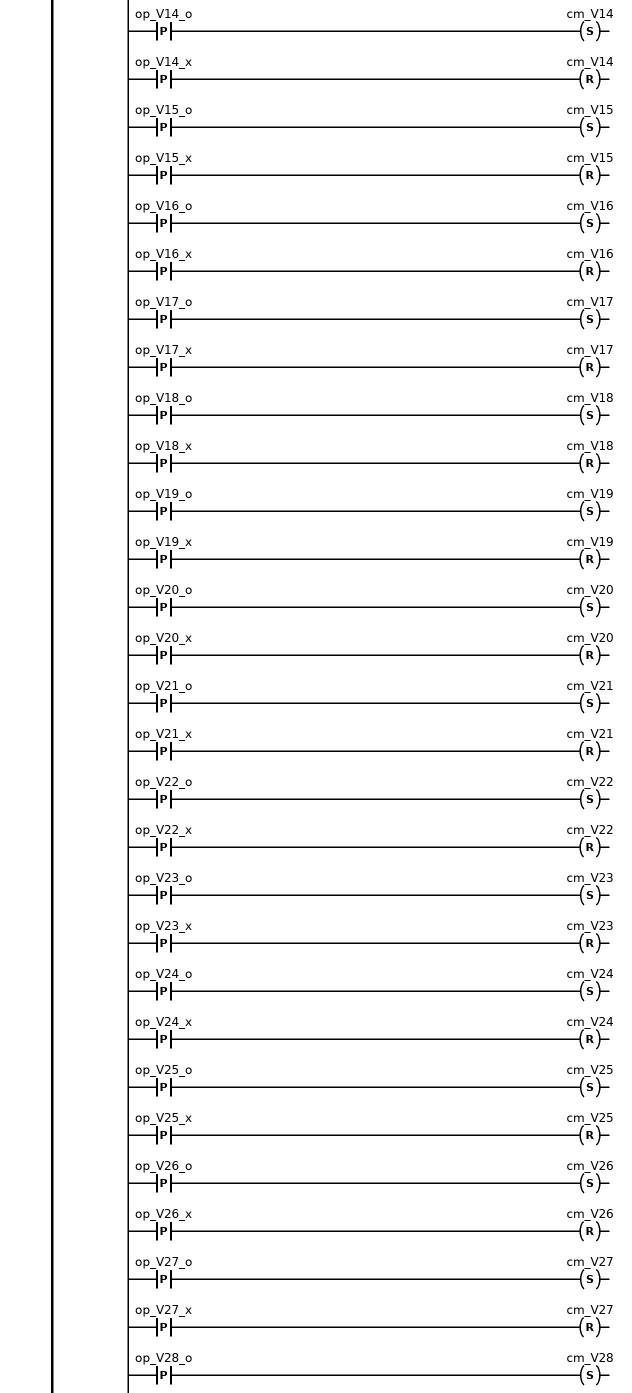
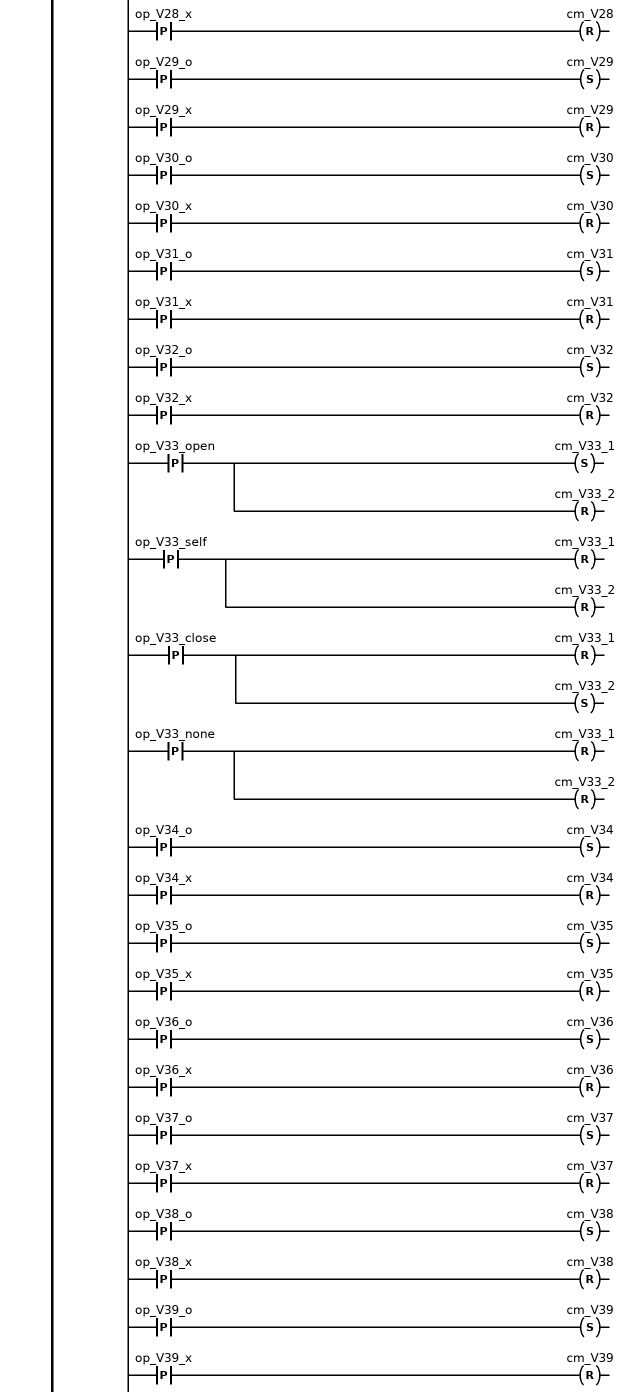
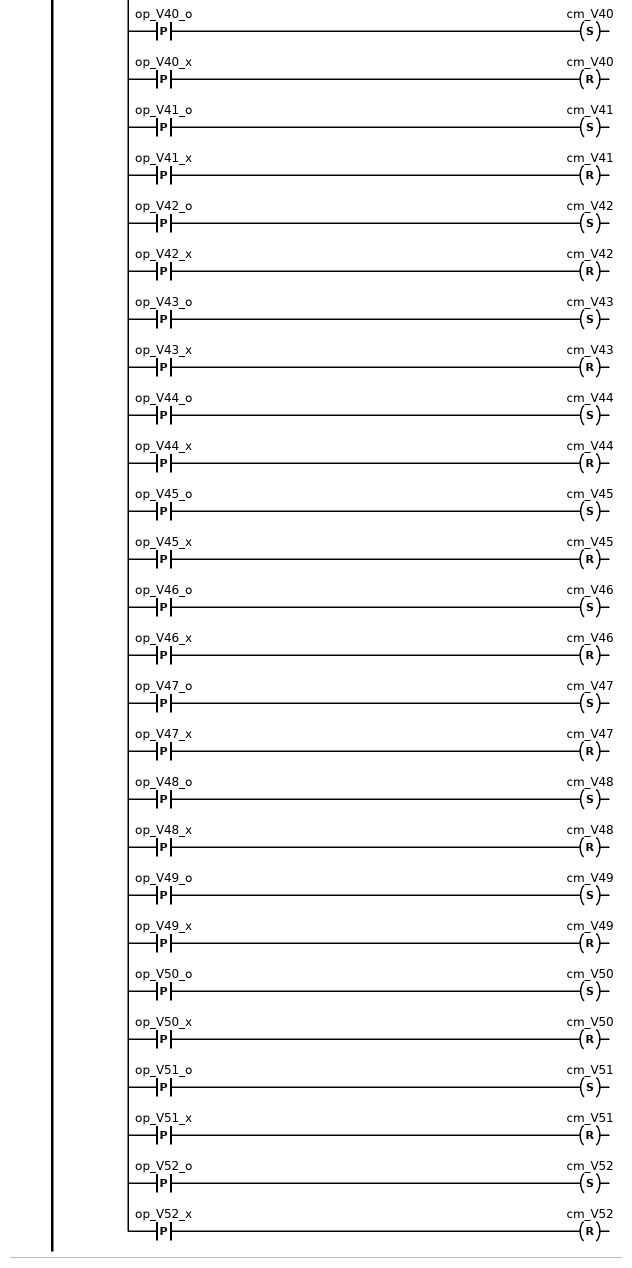
// NETWORK 19
// On/Off CMDS
_w5 := NOT ing_RCP;
_rt113(CLK := op_V01_o);
_w6 := _w5 AND _rt113.Q;
cm_V01 S= _w6;
b_Test S= _w6;
_rt114(CLK := op_V01_x);
_w7 := _w5 AND _rt114.Q;
cm_V01 R= _w7;
b_Test R= _w7;
_rt115(CLK := op_V02_o);
cm_V02 S= _w5 AND _rt115.Q;
_rt116(CLK := op_V02_x);
cm_V02 R= _w5 AND _rt116.Q;
_rt117(CLK := op_V03_o);
cm_V03 S= _w5 AND _rt117.Q;
_rt118(CLK := op_V03_x);
cm_V03 R= _w5 AND _rt118.Q;
_rt119(CLK := op_V04_o);
cm_V04 S= _w5 AND _rt119.Q;
_rt120(CLK := op_V04_x);
cm_V04 R= _w5 AND _rt120.Q;
_rt121(CLK := op_V05_o);
cm_V05 S= _w5 AND _rt121.Q;
_rt122(CLK := op_V05_x);
cm_V05 R= _w5 AND _rt122.Q;
_rt123(CLK := op_V06_o);
cm_V06 S= _w5 AND _rt123.Q;
_rt124(CLK := op_V06_x);
cm_V06 R= _w5 AND _rt124.Q;
_rt125(CLK := op_V07_o);
cm_V07 S= _w5 AND _rt125.Q;
_rt126(CLK := op_V07_x);
cm_V07 R= _w5 AND _rt126.Q;
_rt127(CLK := op_V08_o);
cm_V08 S= _w5 AND _rt127.Q;
_rt128(CLK := op_V08_x);
cm_V08 R= _w5 AND _rt128.Q;
_rt129(CLK := op_V09_o);
cm_V09 S= _w5 AND _rt129.Q;
_rt130(CLK := op_V09_x);
cm_V09 R= _w5 AND _rt130.Q;
_rt131(CLK := op_V10_o);
cm_V10 S= _w5 AND _rt131.Q;
_rt132(CLK := op_V10_x);
cm_V10 R= _w5 AND _rt132.Q;
_rt133(CLK := op_V11_o);
cm_V11 S= _w5 AND _rt133.Q;
_rt134(CLK := op_V11_x);
cm_V11 R= _w5 AND _rt134.Q;
_rt135(CLK := op_V12_o);
cm_V12 S= _w5 AND _rt135.Q;
_rt136(CLK := op_V12_x);
cm_V12 R= _w5 AND _rt136.Q;
_rt137(CLK := op_V13_o);
cm_V13 S= _w5 AND _rt137.Q;
_rt138(CLK := op_V13_x);
cm_V13 R= _w5 AND _rt138.Q;
_rt139(CLK := op_V14_o);
cm_V14 S= _w5 AND _rt139.Q;
_rt140(CLK := op_V14_x);
cm_V14 R= _w5 AND _rt140.Q;
_rt141(CLK := op_V15_o);
cm_V15 S= _w5 AND _rt141.Q;
_rt142(CLK := op_V15_x);
cm_V15 R= _w5 AND _rt142.Q;
_rt143(CLK := op_V16_o);
cm_V16 S= _w5 AND _rt143.Q;
_rt144(CLK := op_V16_x);
cm_V16 R= _w5 AND _rt144.Q;
_rt145(CLK := op_V17_o);
cm_V17 S= _w5 AND _rt145.Q;
_rt146(CLK := op_V17_x);
cm_V17 R= _w5 AND _rt146.Q;
_rt147(CLK := op_V18_o);
cm_V18 S= _w5 AND _rt147.Q;
_rt148(CLK := op_V18_x);
cm_V18 R= _w5 AND _rt148.Q;
_rt149(CLK := op_V19_o);
cm_V19 S= _w5 AND _rt149.Q;
_rt150(CLK := op_V19_x);
cm_V19 R= _w5 AND _rt150.Q;
_rt151(CLK := op_V20_o);
cm_V20 S= _w5 AND _rt151.Q;
_rt152(CLK := op_V20_x);
cm_V20 R= _w5 AND _rt152.Q;
_rt153(CLK := op_V21_o);
cm_V21 S= _w5 AND _rt153.Q;
_rt154(CLK := op_V21_x);
cm_V21 R= _w5 AND _rt154.Q;
_rt155(CLK := op_V22_o);
cm_V22 S= _w5 AND _rt155.Q;
_rt156(CLK := op_V22_x);
cm_V22 R= _w5 AND _rt156.Q;
_rt157(CLK := op_V23_o);
cm_V23 S= _w5 AND _rt157.Q;
_rt158(CLK := op_V23_x);
cm_V23 R= _w5 AND _rt158.Q;
_rt159(CLK := op_V24_o);
cm_V24 S= _w5 AND _rt159.Q;
_rt160(CLK := op_V24_x);
cm_V24 R= _w5 AND _rt160.Q;
_rt161(CLK := op_V25_o);
cm_V25 S= _w5 AND _rt161.Q;
_rt162(CLK := op_V25_x);
cm_V25 R= _w5 AND _rt162.Q;
_rt163(CLK := op_V26_o);
cm_V26 S= _w5 AND _rt163.Q;
_rt164(CLK := op_V26_x);
cm_V26 R= _w5 AND _rt164.Q;
_rt165(CLK := op_V27_o);
cm_V27 S= _w5 AND _rt165.Q;
_rt166(CLK := op_V27_x);
cm_V27 R= _w5 AND _rt166.Q;
_rt167(CLK := op_V28_o);
cm_V28 S= _w5 AND _rt167.Q;
_rt168(CLK := op_V28_x);
cm_V28 R= _w5 AND _rt168.Q;
_rt169(CLK := op_V29_o);
cm_V29 S= _w5 AND _rt169.Q;
_rt170(CLK := op_V29_x);
cm_V29 R= _w5 AND _rt170.Q;
_rt171(CLK := op_V30_o);
cm_V30 S= _w5 AND _rt171.Q;
_rt172(CLK := op_V30_x);
cm_V30 R= _w5 AND _rt172.Q;
_rt173(CLK := op_V31_o);
cm_V31 S= _w5 AND _rt173.Q;
_rt174(CLK := op_V31_x);
cm_V31 R= _w5 AND _rt174.Q;
_rt175(CLK := op_V32_o);
cm_V32 S= _w5 AND _rt175.Q;
_rt176(CLK := op_V32_x);
cm_V32 R= _w5 AND _rt176.Q;
_rt177(CLK := op_V33_open);
_w8 := _w5 AND _rt177.Q;
cm_V33_1 S= _w8;
cm_V33_2 R= _w8;
_rt178(CLK := op_V33_self);
_w9 := _w5 AND _rt178.Q;
cm_V33_1 R= _w9;
cm_V33_2 R= _w9;
_rt179(CLK := op_V33_close);
_w10 := _w5 AND _rt179.Q;
cm_V33_1 R= _w10;
cm_V33_2 S= _w10;
_rt180(CLK := op_V33_none);
_w11 := _w5 AND _rt180.Q;
cm_V33_1 R= _w11;
cm_V33_2 R= _w11;
_rt181(CLK := op_V34_o);
cm_V34 S= _w5 AND _rt181.Q;
_rt182(CLK := op_V34_x);
cm_V34 R= _w5 AND _rt182.Q;
_rt183(CLK := op_V35_o);
cm_V35 S= _w5 AND _rt183.Q;
_rt184(CLK := op_V35_x);
cm_V35 R= _w5 AND _rt184.Q;
_rt185(CLK := op_V36_o);
cm_V36 S= _w5 AND _rt185.Q;
_rt186(CLK := op_V36_x);
cm_V36 R= _w5 AND _rt186.Q;
_rt187(CLK := op_V37_o);
cm_V37 S= _w5 AND _rt187.Q;
_rt188(CLK := op_V37_x);
cm_V37 R= _w5 AND _rt188.Q;
_rt189(CLK := op_V38_o);
cm_V38 S= _w5 AND _rt189.Q;
_rt190(CLK := op_V38_x);
cm_V38 R= _w5 AND _rt190.Q;
_rt191(CLK := op_V39_o);
cm_V39 S= _w5 AND _rt191.Q;
_rt192(CLK := op_V39_x);
cm_V39 R= _w5 AND _rt192.Q;
_rt193(CLK := op_V40_o);
cm_V40 S= _w5 AND _rt193.Q;
_rt194(CLK := op_V40_x);
cm_V40 R= _w5 AND _rt194.Q;
_rt195(CLK := op_V41_o);
cm_V41 S= _w5 AND _rt195.Q;
_rt196(CLK := op_V41_x);
cm_V41 R= _w5 AND _rt196.Q;
_rt197(CLK := op_V42_o);
cm_V42 S= _w5 AND _rt197.Q;
_rt198(CLK := op_V42_x);
cm_V42 R= _w5 AND _rt198.Q;
_rt199(CLK := op_V43_o);
cm_V43 S= _w5 AND _rt199.Q;
_rt200(CLK := op_V43_x);
cm_V43 R= _w5 AND _rt200.Q;
_rt201(CLK := op_V44_o);
cm_V44 S= _w5 AND _rt201.Q;
_rt202(CLK := op_V44_x);
cm_V44 R= _w5 AND _rt202.Q;
_rt203(CLK := op_V45_o);
cm_V45 S= _w5 AND _rt203.Q;
_rt204(CLK := op_V45_x);
cm_V45 R= _w5 AND _rt204.Q;
_rt205(CLK := op_V46_o);
cm_V46 S= _w5 AND _rt205.Q;
_rt206(CLK := op_V46_x);
cm_V46 R= _w5 AND _rt206.Q;
_rt207(CLK := op_V47_o);
cm_V47 S= _w5 AND _rt207.Q;
_rt208(CLK := op_V47_x);
cm_V47 R= _w5 AND _rt208.Q;
_rt209(CLK := op_V48_o);
cm_V48 S= _w5 AND _rt209.Q;
_rt210(CLK := op_V48_x);
cm_V48 R= _w5 AND _rt210.Q;
_rt211(CLK := op_V49_o);
cm_V49 S= _w5 AND _rt211.Q;
_rt212(CLK := op_V49_x);
cm_V49 R= _w5 AND _rt212.Q;
_rt213(CLK := op_V50_o);
cm_V50 S= _w5 AND _rt213.Q;
_rt214(CLK := op_V50_x);
cm_V50 R= _w5 AND _rt214.Q;
_rt215(CLK := op_V51_o);
cm_V51 S= _w5 AND _rt215.Q;
_rt216(CLK := op_V51_x);
cm_V51 R= _w5 AND _rt216.Q;
_rt217(CLK := op_V52_o);
cm_V52 S= _w5 AND _rt217.Q;
_rt218(CLK := op_V52_x);
cm_V52 R= _w5 AND _rt218.Q;

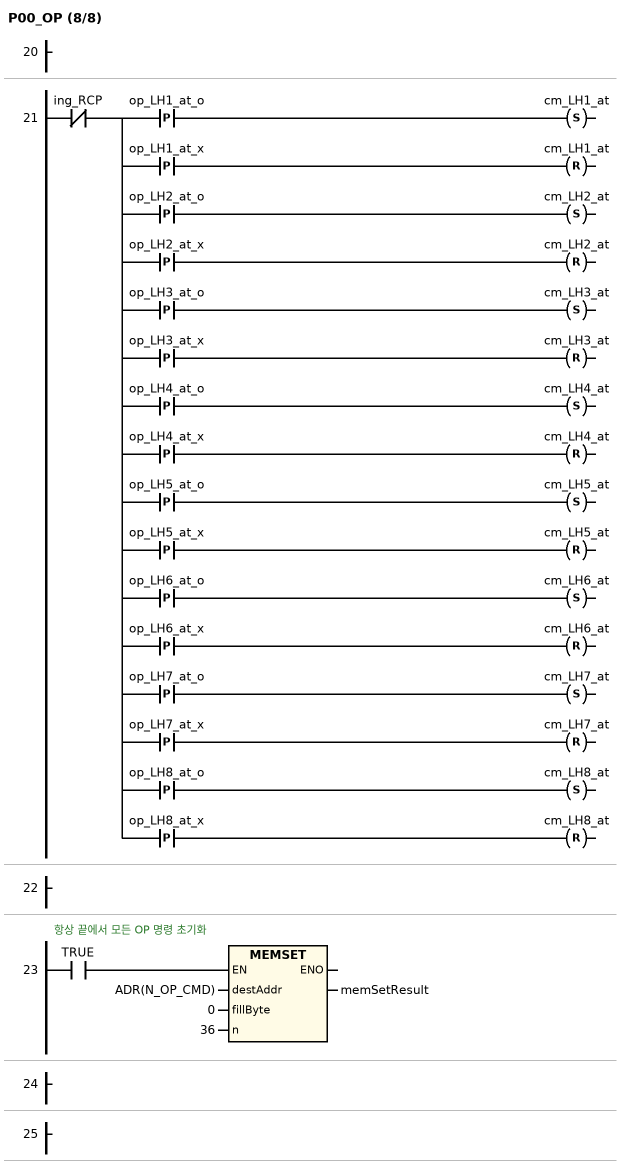
// NETWORK 20

// NETWORK 21
_w12 := NOT ing_RCP;
_rt219(CLK := op_LH1_at_o);
cm_LH1_at S= _w12 AND _rt219.Q;
_rt220(CLK := op_LH1_at_x);
cm_LH1_at R= _w12 AND _rt220.Q;
_rt221(CLK := op_LH2_at_o);
cm_LH2_at S= _w12 AND _rt221.Q;
_rt222(CLK := op_LH2_at_x);
cm_LH2_at R= _w12 AND _rt222.Q;
_rt223(CLK := op_LH3_at_o);
cm_LH3_at S= _w12 AND _rt223.Q;
_rt224(CLK := op_LH3_at_x);
cm_LH3_at R= _w12 AND _rt224.Q;
_rt225(CLK := op_LH4_at_o);
cm_LH4_at S= _w12 AND _rt225.Q;
_rt226(CLK := op_LH4_at_x);
cm_LH4_at R= _w12 AND _rt226.Q;
_rt227(CLK := op_LH5_at_o);
cm_LH5_at S= _w12 AND _rt227.Q;
_rt228(CLK := op_LH5_at_x);
cm_LH5_at R= _w12 AND _rt228.Q;
_rt229(CLK := op_LH6_at_o);
cm_LH6_at S= _w12 AND _rt229.Q;
_rt230(CLK := op_LH6_at_x);
cm_LH6_at R= _w12 AND _rt230.Q;
_rt231(CLK := op_LH7_at_o);
cm_LH7_at S= _w12 AND _rt231.Q;
_rt232(CLK := op_LH7_at_x);
cm_LH7_at R= _w12 AND _rt232.Q;
_rt233(CLK := op_LH8_at_o);
cm_LH8_at S= _w12 AND _rt233.Q;
_rt234(CLK := op_LH8_at_x);
cm_LH8_at R= _w12 AND _rt234.Q;

// NETWORK 22

// NETWORK 23
// 항상 끝에서 모든 OP 명령 초기화
memSetResult := MEMSET(destAddr := ADR(N_OP_CMD), fillByte := 0, n := 36);

// NETWORK 24

// NETWORK 25

END_PROGRAM

// ---- POUs/MR_PRG/P01_Init_N_Retain.TcPOU
PROGRAM P01_Init_N_Retain
VAR RETAIN
    R_LH_TB_SV: ARRAY[0..14] OF REAL;

	R_SOL_IDX1: ARRAY[0..31] OF SINT;	
	R_SOL_IDX2: ARRAY[0..31] OF SINT;
	
	R_ETC_A: ARRAY[0..19] OF REAL;
	R_ETC_D: ARRAY[0..19] OF BOOL;
				
	R_EN_RAMP: ARRAY[0..29] OF BOOL;
	R_EN_RCP_RAMP: ARRAY[0..29] OF BOOL;
	
	R_EN_AL: ARRAY[0..143] OF BOOL;
	R_Dev_AL: ARRAY[0..29] OF WORD;	
	R_DevTM_AL: ARRAY[0..29] OF WORD;
	R_A_SV_AL: ARRAY[0..19] OF REAL; 	//Alarm analog check SV	
	
	R_EN_WN: ARRAY[0..63] OF BOOL;
	R_Dev_WN: ARRAY[0..29] OF WORD;	
	R_DevTM_WN: ARRAY[0..29] OF WORD;
	R_A_SV_WN: ARRAY[0..19] OF REAL;	//Warn analog check SV
	
	R_MIN: ARRAY[0..69] OF REAL; 
	R_MAX: ARRAY[0..69] OF REAL; 	
		
	R_US_D: ARRAY[0..3, 0..29] OF BYTE;	//User State - Digital
	R_US_A: ARRAY[0..3, 0..31] OF REAL; 	//User State - Analog 
	R_US_A_EN: ARRAY[0..3, 0..31] OF BOOL; 	//User State - Analog EN 
	
	R_MS_SET: ARRAY[0..5, 0..9] OF REAL; 	//Mo Source Set
	R_PV_ROT_INCH_PLS: REAL; 
	R_PV_ROT_1TURN_PLS: REAL;

    R_TV_posMode: BOOL; 	
END_VAR

VAR
	T1 : Ton := (PT:=T#1S);//dats save Timer
	idx, idx2 : DINT;
	cmp_RTM_UNIT : UINT;
	cmp_RTM_UNIT_STEPS : UINT;
END_VAR


T1(IN:= 1);

IF is_TCAT_started = 0 THEN	
	MEMMOVE(destAddr:=ADR(N_LH_TB_SV), srcAddr:=ADR(R_LH_TB_SV), n:=SIZEOF(N_LH_TB_SV));
	
	MEMMOVE(destAddr:=ADR(N_SOL1), srcAddr:=ADR(R_SOL_IDX1), n:=SIZEOF(N_SOL1));
	MEMMOVE(destAddr:=ADR(N_SOL2), srcAddr:=ADR(R_SOL_IDX2), n:=SIZEOF(N_SOL2));
	
	MEMMOVE(destAddr:=ADR(N_ETC_A), srcAddr:=ADR(R_ETC_A), n:=SIZEOF(N_ETC_A));
	MEMMOVE(destAddr:=ADR(N_ETC_D), srcAddr:=ADR(R_ETC_D), n:=SIZEOF(N_ETC_D));
	
	MEMMOVE(destAddr:=ADR(N_EN_RAMP), srcAddr:=ADR(R_EN_RAMP), n:=SIZEOF(N_EN_RAMP)); 
	MEMMOVE(destAddr:=ADR(N_EN_RCP_RAMP), srcAddr:=ADR(R_EN_RCP_RAMP), n:=SIZEOF(N_EN_RCP_RAMP));
	
	MEMMOVE(destAddr:=ADR(N_EN_AL), srcAddr:=ADR(R_EN_AL), n:=SIZEOF(N_EN_AL));		
	MEMMOVE(destAddr:=ADR(N_Dev_AL), srcAddr:=ADR(R_Dev_AL), n:=SIZEOF(N_Dev_AL));
	MEMMOVE(destAddr:=ADR(N_DevTM_AL), srcAddr:=ADR(R_DevTM_AL), n:=SIZEOF(N_DevTM_AL));	
	MEMMOVE(destAddr:=ADR(N_A_SV_AL), srcAddr:=ADR(R_A_SV_AL), n:=SIZEOF(N_A_SV_AL));
	
	MEMMOVE(destAddr:=ADR(N_EN_WN), srcAddr:=ADR(R_EN_WN), n:=SIZEOF(N_EN_WN));	
	MEMMOVE(destAddr:=ADR(N_Dev_WN), srcAddr:=ADR(R_Dev_WN), n:=SIZEOF(N_Dev_WN));
	MEMMOVE(destAddr:=ADR(N_DevTM_WN), srcAddr:=ADR(R_DevTM_WN), n:=SIZEOF(N_DevTM_WN));
	MEMMOVE(destAddr:=ADR(N_A_SV_WN), srcAddr:=ADR(R_A_SV_WN), n:=SIZEOF(N_A_SV_WN));	
		
	MEMMOVE(destAddr:=ADR(N_MIN), srcAddr:=ADR(R_MIN), n:=SIZEOF(N_MIN));
	MEMMOVE(destAddr:=ADR(N_MAX), srcAddr:=ADR(R_MAX), n:=SIZEOF(N_MAX));
   
	MEMMOVE(destAddr:=ADR(N_US_D), srcAddr:=ADR(R_US_D), n:=SIZEOF(N_US_D));
	MEMMOVE(destAddr:=ADR(N_US_A), srcAddr:=ADR(R_US_A), n:=SIZEOF(N_US_A));
	MEMMOVE(destAddr:=ADR(N_US_A_EN), srcAddr:=ADR(R_US_A_EN), n:=SIZEOF(N_US_A_EN));	
              
	MEMMOVE(destAddr:=ADR(N_MS_SET), srcAddr:=ADR(R_MS_SET), n:=SIZEOF(N_MS_SET));
   
	pv_ROT_inchPulse := R_PV_ROT_INCH_PLS;  
	pv_ROT_1turnPulse := 0;//PV_ROT_1TURN_PLS; 

    en_TV_posMode := R_TV_posMode; 
      
   //Default Value Check
  	ACT_Default_Value_Check();
	
	IF e_RTM_UNIT < 100 THEN e_RTM_UNIT := 100; END_IF
	IF e_RTM_UNIT_STEPS < 1 THEN e_RTM_UNIT_STEPS := 1; END_IF        	
	cmp_RTM_UNIT := e_RTM_UNIT ;
	cmp_RTM_UNIT_STEPS := e_RTM_UNIT_STEPS;
	RTM_UNIT := UINT_TO_TIME(e_RTM_UNIT / e_RTM_UNIT_STEPS);
		
	pv_US := -1;	
	IF e_US_START > 0 THEN
		CASE e_US_START OF
			1: cm_US1 := 1;
			2: cm_US2 := 1;
			3: cm_US3 := 1;
			4: cm_US4 := 1;
		END_CASE
	END_IF
	//tsv_Pres := sv_PRES:= 760;
	//rtm_Pres := 0;	
    ing_MAINT := 0;
END_IF

IF T1.Q AND is_TCAT_started = 0 THEN
	is_TCAT_started := 1;
END_IF


//변경되는 Retain Data 저장
IF is_TCAT_started THEN
	//always save
	IF T1.Q THEN
		MEMMOVE(destAddr:=ADR(R_LH_TB_SV), srcAddr:=ADR(N_LH_TB_SV), n:=SIZEOF(N_LH_TB_SV));
	END_IF	

	//SOL INDEX1 Data
   IF cm_SOL1_save THEN
		MEMMOVE(destAddr:=ADR(R_SOL_IDX1), srcAddr:=ADR(N_SOL1), n:=SIZEOF(N_SOL1));
	   cm_SOL1_save := 0;
   END_IF
   
   	//SOL INDEX2 Data
   IF cm_SOL2_save THEN
		MEMMOVE(destAddr:=ADR(R_SOL_IDX2), srcAddr:=ADR(N_SOL2), n:=SIZEOF(N_SOL2));
	   cm_SOL2_save := 0;
   END_IF

   //Etc System Data
   IF cm_ETC_save THEN
		MEMMOVE(destAddr:=ADR(R_ETC_A), srcAddr:=ADR(N_ETC_A), n:=SIZEOF(N_ETC_A));
		MEMMOVE(destAddr:=ADR(R_ETC_D), srcAddr:=ADR(N_ETC_D), n:=SIZEOF(N_ETC_D));
		cm_ETC_save := 0;
   END_IF

   IF cm_EN_RAMP_save THEN
	   MEMMOVE(destAddr:=ADR(R_EN_RAMP), srcAddr:=ADR(N_EN_Ramp), n:=SIZEOF(N_EN_Ramp));
	   MEMMOVE(destAddr:=ADR(R_EN_RCP_RAMP), srcAddr:=ADR(N_EN_RCP_RAMP), n:=SIZEOF(N_EN_RCP_RAMP));
	   cm_EN_RAMP_save := 0;
   END_IF

   //Alarm Data
   IF cm_AL_save THEN
	   MEMMOVE(destAddr:=ADR(R_EN_AL), srcAddr:=ADR(N_EN_AL), n:=SIZEOF(N_EN_AL));
	   MEMMOVE(destAddr:=ADR(R_Dev_AL), srcAddr:=ADR(N_Dev_AL), n:=SIZEOF(N_Dev_AL));
	   MEMMOVE(destAddr:=ADR(R_DevTM_AL), srcAddr:=ADR(N_DevTM_AL), n:=SIZEOF(N_DevTM_AL));
	   MEMMOVE(destAddr:=ADR(R_A_SV_AL), srcAddr:=ADR(N_A_SV_AL), n:=SIZEOF(N_A_SV_AL));
   	   cm_AL_save := 0;
   END_IF
   
   //Warning Data
   IF cm_WN_save THEN
	   MEMMOVE(destAddr:=ADR(R_EN_WN), srcAddr:=ADR(N_EN_WN), n:=SIZEOF(N_EN_WN));
	   MEMMOVE(destAddr:=ADR(R_Dev_WN), srcAddr:=ADR(N_Dev_WN), n:=SIZEOF(N_Dev_WN));
	   MEMMOVE(destAddr:=ADR(R_DevTM_WN), srcAddr:=ADR(N_DevTM_WN), n:=SIZEOF(N_DevTM_WN));
	   MEMMOVE(destAddr:=ADR(R_A_SV_WN), srcAddr:=ADR(N_A_SV_WN), n:=SIZEOF(N_A_SV_WN));      
   	   cm_WN_save := 0;
   END_IF    
         
	//Max Value
   IF cm_MAX_save THEN
	   MEMMOVE(destAddr:=ADR(R_MIN), srcAddr:=ADR(N_MIN), n:=SIZEOF(N_MIN));
	   MEMMOVE(destAddr:=ADR(R_MAX), srcAddr:=ADR(N_MAX), n:=SIZEOF(N_MAX));
	   cm_MAX_save := 0;
   END_IF
   
   //User State
   IF cm_US_save THEN
	   MEMMOVE(destAddr:=ADR(R_US_D), srcAddr:=ADR(N_US_D), n:=SIZEOF(N_US_D));
	   MEMMOVE(destAddr:=ADR(R_US_A), srcAddr:=ADR(N_US_A), n:=SIZEOF(N_US_A));
	   MEMMOVE(destAddr:=ADR(R_US_A_EN), srcAddr:=ADR(N_US_A_EN), n:=SIZEOF(N_US_A_EN));
	   cm_US_save := 0;
   END_IF
               	        
   	//Mo Source Weight init
	IF cm_MO_save THEN
		MEMMOVE(destAddr:=ADR(R_MS_SET), srcAddr:=ADR(N_MS_SET), n:=SIZEOF(N_MS_SET));
	   	cm_MO_save := 0;
	ELSE//Always Save
		IF T1.Q THEN
			FOR idx := 0 TO 5 DO
				FOR idx2 := 0 TO 9 DO
					R_MS_SET[idx, idx2] := N_MS_SET[idx, idx2];
				END_FOR
			END_FOR
		END_IF  	   
   	END_IF

   	//Rotation Pulse Total Sum
   	R_PV_ROT_INCH_PLS := pv_ROT_inchPulse; 
	R_PV_ROT_1TURN_PLS := pv_ROT_1turnPulse;
            
	IF (cmp_RTM_UNIT <> e_RTM_UNIT) OR (cmp_RTM_UNIT_STEPS <> e_RTM_UNIT_STEPS) THEN
		cmp_RTM_UNIT := e_RTM_UNIT;
		cmp_RTM_UNIT_STEPS := e_RTM_UNIT_STEPS;
		RTM_UNIT := UINT_TO_TIME(e_RTM_UNIT / e_RTM_UNIT_STEPS);   
	END_IF 

	IF cm_TV_presMode THEN
		en_TV_posMode := R_TV_posMode := 0;
		cm_TV_presMode := 0;
	END_IF  

	IF cm_TV_posMode THEN
	  	en_TV_posMode := R_TV_posMode := 1;
		cm_TV_posMode := 0;
	END_IF   
END_IF;


IF T1.Q THEN
	T1(IN:= 0);
END_IF

ACTION ACT_Default_Value_Check:
   //Default Value Check
   IF e_ROT_AO_SLOPE_FACTOR = 0 THEN
	   e_ROT_AO_SLOPE_FACTOR := 1;
   END_IF
   IF e_ROT_SLOW_RPM = 0 THEN
	   e_ROT_SLOW_RPM := 1;
   END_IF
   IF e_ROT_60_RPM = 0 THEN
	   e_ROT_60_RPM := 1;
   END_IF
   IF e_ROT_60_PT = 0 THEN
	   e_ROT_60_PT := 750;
   END_IF
END_ACTION

END_PROGRAM

// ---- POUs/MR_PRG/P02_Init_MC.TcPOU
PROGRAM P02_Init_MC
VAR
	p_Start: R_TRIG;
	nCase: INT := 0;
	T1: TON := (PT:= T#5S);
END_VAR

//IF s_is_All_MC_on THEN
	//RETURN;
//END_IF

//Start
IF ing_MAINT = 0 AND s_CM_ALL_MC_ON = 0 AND s_is_All_MC_on = 0 THEN
	s_CM_ALL_MC_ON := 1;
END_IF


T1(IN:= nCase > 0);
p_Start(CLK:= s_CM_ALL_MC_ON AND s_is_All_MC_on = 0);

IF p_Start.Q THEN
	nCase := 1;
END_IF

CASE nCase OF
	1://IH MC
	    IF do_IH_mc THEN
			nCase := 11;
		ELSE
			T1(IN:= 0);
			cm_IH_mc := 1;			
			nCase := 2;
		END_IF
	2://wait
		IF T1.Q AND do_IH_mc THEN
			T1(IN:= 0);
			nCase := 11;
		END_IF
	11://TB_mc
	    IF do_TB_mc THEN
			nCase := 21;
		ELSE
			T1(IN:= 0);
			cm_TB_mc := 1;			
			nCase := 12;
		END_IF
	12://wait
		IF T1.Q AND do_TB_mc THEN
			T1(IN:= 0);
			nCase := 21;
		END_IF
	21://VP_mc
	    IF do_VP_mc THEN
			nCase := 31;
		ELSE
			T1(IN:= 0);
			cm_VP_mc := 1;			
			nCase := 22;
		END_IF
	22://wait
		IF T1.Q AND do_VP_mc THEN
			T1(IN:= 0);
			nCase := 31;
		END_IF
	31://LH_mc
	    IF do_LH_mc THEN
			nCase := 100;
		ELSE
			T1(IN:= 0);
			cm_LH_mc := 1;			
			nCase := 32;
		END_IF
	32://wait
		IF T1.Q AND do_LH_mc THEN
			T1(IN:= 0);
			nCase := 100;
		END_IF
	100://End
		s_CM_ALL_MC_ON := 0;
		nCase := 0;		
END_CASE

s_is_All_MC_on := do_IH_mc AND do_TB_mc AND do_VP_mc AND do_LH_mc;

END_PROGRAM

// ---- POUs/P02_P2P/P02_P2P.TcPOU
PROGRAM P02_P2P
VAR
END_VAR

//P2P_ST300_MODBUS();
P2P_LH();
P2P_TB();

END_PROGRAM

// ---- POUs/P02_P2P/P2P_LH.TcPOU
PROGRAM P2P_LH
VAR
	LH1_sv, LH2_sv, LH3_sv, LH4_sv, LH5_sv, LH6_sv, LH7_sv, LH8_sv: REAL := 0;
	LH1_at, LH2_at, LH3_at, LH4_at, LH5_at, LH6_at, LH7_at, LH8_at: BOOL := 0;
	
	T_TMOut: TON := (PT:=T#1S);
	iStep: INT := 1;
	bTx_en: BOOL;
	bTx_ok: BOOL;
	p2p_mode: INT; //1 = PV Req, 2 = STATUS Req, 3 = SV Write, 4 = AT On/Off
	p2p_cnt1, p2p_cnt2, p2p_cnt3, p2p_cnt4: INT := 0;
	
	addrMin: INT := 1;
	addrMax: INT := 8;
	
	//For Send
	T_Tx: TON := (PT:=T#10MS);
	fbTx: SendString;
	strTx: STRING;
	bTx_busy: BOOL;
	eTx_errID: ComError_t;	
			
	//For Receive
	T_Rx: TON := (PT:=T#10MS);
	bRx_ok: BOOL;	
	fbRx: ReceiveString;
	strRx: STRING;
	bRx_received: BOOL;
	bRx_busy: BOOL;
	eRx_errID: ComError_t;
	bRx_tmout: BOOL;
	strHex: STRING;	
		
	iPvDecimal: INT := 1;// Config Data
END_VAR

//LH: Line Heater x 8EA -> 8Channel TIC 1EA
//Maker: HANYOUNG NUX
//Model: MC9-8RD0SS32
//Temp Range: -15 ~200℃
//RS485: 9600, DataBit(8), Parity(None), StopBit(1)
//BCC Check X

IF bTx_en = Off THEN
	bTx_en := 1;
	bTx_ok := bRx_ok := 0;
		
	IF p2p_mode <> 1 THEN //PV Req
		strTx := '$0201DRS,08,0001$0D$0A';
		p2p_mode := 1;
	ELSE //STATUS Req
		strTx := '$0201DRS,08,0111$0D$0A';
		p2p_mode := 2;
	END_IF
	
	//SV Change Check -> SV Write Mode
	IF LH1_sv <> sv_LH1 THEN
		LH1_sv := sv_LH1;
		strTx := CONCAT(CONCAT('$0201DWR,03,0301,0001,0302,0001,0401,', F_LH_SV(SV:= LH1_sv, nDecimal:= iPvDecimal)), '$0D$0A'); //0301(ZONE_NO),0001(ZONE_1),0302(CH_NO),0001(CH_1),0401(SV)		
		p2p_mode := 3;	
	ELSIF LH2_sv <> sv_LH2 THEN
		LH2_sv := sv_LH2;
		strTx := CONCAT(CONCAT('$0201DWR,03,0301,0001,0302,0002,0401,', F_LH_SV(SV:= LH2_sv, nDecimal:= iPvDecimal)), '$0D$0A'); //0301(ZONE_NO),0001(ZONE_1),0302(CH_NO),0002(CH_2),0401(SV)		
		p2p_mode := 3;		
	ELSIF LH3_sv <> sv_LH3 THEN
		LH3_sv := sv_LH3;
		strTx := CONCAT(CONCAT('$0201DWR,03,0301,0001,0302,0003,0401,', F_LH_SV(SV:= LH3_sv, nDecimal:= iPvDecimal)), '$0D$0A'); //0301(ZONE_NO),0001(ZONE_1),0302(CH_NO),0002(CH_3),0401(SV)		
		p2p_mode := 3;		
	ELSIF LH4_sv <> sv_LH4 THEN
		LH4_sv := sv_LH4;
		strTx := CONCAT(CONCAT('$0201DWR,03,0301,0001,0302,0004,0401,', F_LH_SV(SV:= LH4_sv, nDecimal:= iPvDecimal)), '$0D$0A'); //0301(ZONE_NO),0001(ZONE_1),0302(CH_NO),0002(CH_4),0401(SV)		
		p2p_mode := 3;		
	ELSIF LH5_sv <> sv_LH5 THEN
		LH5_sv := sv_LH5;
		strTx := CONCAT(CONCAT('$0201DWR,03,0301,0001,0302,0005,0401,', F_LH_SV(SV:= LH5_sv, nDecimal:= iPvDecimal)), '$0D$0A'); //0301(ZONE_NO),0001(ZONE_1),0302(CH_NO),0002(CH_5),0401(SV)		
		p2p_mode := 3;		
	ELSIF LH6_sv <> sv_LH6 THEN
		LH6_sv := sv_LH6;
		strTx := CONCAT(CONCAT('$0201DWR,03,0301,0001,0302,0006,0401,', F_LH_SV(SV:= LH6_sv, nDecimal:= iPvDecimal)), '$0D$0A'); //0301(ZONE_NO),0001(ZONE_1),0302(CH_NO),0002(CH_6),0401(SV)		
		p2p_mode := 3;	
	ELSIF LH7_sv <> sv_LH7 THEN
		LH7_sv := sv_LH7;
		strTx := CONCAT(CONCAT('$0201DWR,03,0301,0001,0302,0007,0401,', F_LH_SV(SV:= LH7_sv, nDecimal:= iPvDecimal)), '$0D$0A'); //0301(ZONE_NO),0001(ZONE_1),0302(CH_NO),0002(CH_7),0401(SV)		
		p2p_mode := 3;	
	ELSIF LH8_sv <> sv_LH8 THEN
		LH8_sv := sv_LH8;
		strTx := CONCAT(CONCAT('$0201DWR,03,0301,0001,0302,0008,0401,', F_LH_SV(SV:= LH8_sv, nDecimal:= iPvDecimal)), '$0D$0A'); //0301(ZONE_NO),0001(ZONE_1),0302(CH_NO),0002(CH_8),0401(SV)		
		p2p_mode := 3;	
	
	ELSIF LH1_at <> cm_LH1_at THEN//AT
		LH1_at := cm_LH1_at;
		IF LH1_at THEN	strTx := '$0201DWR,02,0302,0001,0501,0001$0D$0A'; 		 //0302(CH_NO),0001(CH_1),0501(AT),0001(AT-ON)
        ELSE			strTx := '$0201DWR,02,0302,0001,0501,0000$0D$0A'; END_IF//0302(CH_NO),0001(CH_1),0501(AT),0001(AT-OFF)		
		p2p_mode := 4;//AT Mode
	ELSIF LH2_at <> cm_LH2_at THEN//AT
		LH2_at := cm_LH2_at;
		IF LH2_at THEN	strTx := '$0201DWR,02,0302,0002,0501,0001$0D$0A'; 		 //0302(CH_NO),0002(CH_2),0501(AT),0001(AT-ON)
        ELSE			strTx := '$0201DWR,02,0302,0002,0501,0000$0D$0A'; END_IF//0302(CH_NO),0002(CH_2),0501(AT),0001(AT-OFF)		
		p2p_mode := 4;//AT Mode
	ELSIF LH3_at <> cm_LH3_at THEN//AT
		LH3_at := cm_LH3_at;
		IF LH3_at THEN	strTx := '$0201DWR,02,0302,0003,0501,0001$0D$0A'; 		 //0302(CH_NO),0003(CH_3),0501(AT),0001(AT-ON)
        ELSE			strTx := '$0201DWR,02,0302,0003,0501,0000$0D$0A'; END_IF//0302(CH_NO),0003(CH_3),0501(AT),0001(AT-OFF)		
		p2p_mode := 4;//AT Mode
	ELSIF LH4_at <> cm_LH4_at THEN//AT
		LH4_at := cm_LH4_at;
		IF LH4_at THEN	strTx := '$0201DWR,02,0302,0004,0501,0001$0D$0A'; 		 //0302(CH_NO),0004(CH_4),0501(AT),0001(AT-ON)
        ELSE			strTx := '$0201DWR,02,0302,0004,0501,0000$0D$0A'; END_IF//0302(CH_NO),0004(CH_4),0501(AT),0001(AT-OFF)		
		p2p_mode := 4;//AT Mode
	ELSIF LH5_at <> cm_LH5_at THEN//AT
		LH5_at := cm_LH5_at;
		IF LH5_at THEN	strTx := '$0201DWR,02,0302,0005,0501,0001$0D$0A'; 		 //0302(CH_NO),0005(CH_5),0501(AT),0001(AT-ON)
        ELSE			strTx := '$0201DWR,02,0302,0005,0501,0000$0D$0A'; END_IF//0302(CH_NO),0005(CH_5),0501(AT),0001(AT-OFF)		
		p2p_mode := 4;//AT Mode
	ELSIF LH6_at <> cm_LH6_at THEN//AT
		LH6_at := cm_LH6_at;
		IF LH6_at THEN	strTx := '$0201DWR,02,0302,0006,0501,0001$0D$0A'; 		 //0302(CH_NO),0006(CH_6),0501(AT),0001(AT-ON)
        ELSE			strTx := '$0201DWR,02,0302,0006,0501,0000$0D$0A'; END_IF//0302(CH_NO),0006(CH_6),0501(AT),0001(AT-OFF)		
		p2p_mode := 4;//AT Mode
	ELSIF LH7_at <> cm_LH7_at THEN//AT
		LH7_at := cm_LH7_at;
		IF LH7_at THEN	strTx := '$0201DWR,02,0302,0007,0501,0001$0D$0A'; 		 //0302(CH_NO),0007(CH_7),0501(AT),0001(AT-ON)
        ELSE			strTx := '$0201DWR,02,0302,0007,0501,0000$0D$0A'; END_IF//0302(CH_NO),0007(CH_7),0501(AT),0001(AT-OFF)		
		p2p_mode := 4;//AT Mode
	ELSIF LH8_at <> cm_LH8_at THEN//AT
		LH8_at := cm_LH8_at;
		IF LH8_at THEN	strTx := '$0201DWR,02,0302,0008,0501,0001$0D$0A'; 		 //0302(CH_NO),0008(CH_8),0501(AT),0001(AT-ON)
        ELSE			strTx := '$0201DWR,02,0302,0008,0501,0000$0D$0A'; END_IF//0302(CH_NO),0008(CH_8),0501(AT),0001(AT-OFF)		
		p2p_mode := 4;//AT Mode
	END_IF
	
END_IF


//Tx
T_Tx(IN:=bTx_en AND bTx_ok = 0);
IF T_Tx.Q OR fbTx.Busy THEN
	bTx_ok := 1;	
	fbTx(SendString:= strTx, TXbuffer:= TxBuf_LH, Busy=> bTx_busy, Error=> );	
	IF fbTx.Error <> COMERROR_NOERROR THEN
		eTx_errID := fbTx.Error;
		bTx_ok := 0;
	ELSE
		eTx_errID := COMERROR_NOERROR;
		bTx_ok := 1;					
	END_IF
END_IF

//Rx
fbRx(Prefix:= '$02', Suffix:= '$0D$0A',
	Timeout:= T#1S, ReceivedString:= strRx,
	RXbuffer:= RxBuf_LH, StringReceived=> bRx_received,
	Busy=> bRx_busy, Error=> eRx_errID,
	RxTimeout=> bRx_tmout);
	
IF bRx_received THEN
	bRx_received := 0;
	bRx_ok := 1;		
	//Read PV
	IF p2p_mode = 1 THEN //1 = PV Req		
		strHex := MID(STR:=strRx, LEN:=4, POS:=11); //'$0201DRS,OK,1900,1900,1900,1900,1900,1900,1900,1900$R$N' '$0D$0A' == '$R$N' 		
		pv_LH1 := F_LH_PV(hexPV:= strHex, nDecimal:= iPvDecimal);
		strHex := MID(STR:=strRx, LEN:=4, POS:=16); 
		pv_LH2 := F_LH_PV(hexPV:= strHex, nDecimal:= iPvDecimal);
		strHex := MID(STR:=strRx, LEN:=4, POS:=21); 
		pv_LH3 := F_LH_PV(hexPV:= strHex, nDecimal:= iPvDecimal);
		strHex := MID(STR:=strRx, LEN:=4, POS:=26); 
		pv_LH4 := F_LH_PV(hexPV:= strHex, nDecimal:= iPvDecimal);
		strHex := MID(STR:=strRx, LEN:=4, POS:=31); 
		pv_LH5 := F_LH_PV(hexPV:= strHex, nDecimal:= iPvDecimal);
		strHex := MID(STR:=strRx, LEN:=4, POS:=36); 
		pv_LH6 := F_LH_PV(hexPV:= strHex, nDecimal:= iPvDecimal);
		strHex := MID(STR:=strRx, LEN:=4, POS:=41); 
		pv_LH7 := F_LH_PV(hexPV:= strHex, nDecimal:= iPvDecimal);
		strHex := MID(STR:=strRx, LEN:=4, POS:=46); 
		pv_LH8 := F_LH_PV(hexPV:= strHex, nDecimal:= iPvDecimal);
		p2p_cnt1 := p2p_cnt1 + 1;
	ELSIF p2p_mode = 2 THEN //2 = STATUS Req			
		strHex := MID(STR:=strRx, LEN:=4, POS:=11); //'$0201DRS,OK,1900,1900,1900,1900,1900,1900,1900,1900$R$N' '$0D$0A' == '$R$N' 		
		is_LH1_run := strHex = '0002';
		is_LH1_at := strHex = '0004';
		is_LH1_err := strHex = '0080';
		strHex := MID(STR:=strRx, LEN:=4, POS:=16); 
		is_LH2_run := strHex = '0002';
		is_LH2_at := strHex = '0004';
		is_LH2_err := strHex = '0080';
		strHex := MID(STR:=strRx, LEN:=4, POS:=21); 
		is_LH3_run := strHex = '0002';
		is_LH3_at := strHex = '0004';
		is_LH3_err := strHex = '0080';
		strHex := MID(STR:=strRx, LEN:=4, POS:=26); 
		is_LH4_run := strHex = '0002';
		is_LH4_at := strHex = '0004';
		is_LH4_err := strHex = '0080';
		strHex := MID(STR:=strRx, LEN:=4, POS:=31); 
		is_LH5_run := strHex = '0002';
		is_LH5_at := strHex = '0004';
		is_LH5_err := strHex = '0080';
		strHex := MID(STR:=strRx, LEN:=4, POS:=36); 
		is_LH6_run := strHex = '0002';
		is_LH6_at := strHex = '0004';
		is_LH6_err := strHex = '0080';
		strHex := MID(STR:=strRx, LEN:=4, POS:=41); 
		is_LH7_run := strHex = '0002';
		is_LH7_at := strHex = '0004';
		is_LH7_err := strHex = '0080';
		strHex := MID(STR:=strRx, LEN:=4, POS:=46); 
		is_LH8_run := strHex = '0002';
		is_LH8_at := strHex = '0004';
		is_LH8_err := strHex = '0080';
		p2p_cnt2 := p2p_cnt2 + 1;
	ELSIF p2p_mode = 3 THEN //3 = SV Write
		p2p_cnt3 := p2p_cnt3 + 1;
	ELSIF p2p_mode = 4 THEN //4 = AT On/Off
		p2p_cnt4 := p2p_cnt4 + 1;		
	END_IF
END_IF
	
//Next LH
T_Rx(IN:= bRx_ok);
T_TMOut(IN:= 1);
IF T_Rx.Q OR T_TMOut.Q THEN
	T_Rx(IN:= 0);
	T_TMOut(IN:= 0);
	bTx_en := 0;
	IF iStep < addrMax THEN	
		iStep := iStep + 1;
	ELSE					
		iStep := addrMin; 
	END_IF
END_IF

END_PROGRAM

// ---- POUs/P02_P2P/P2P_TB.TcPOU
PROGRAM P2P_TB
VAR
    TB1_SV, TB2_SV, TB3_SV, TB4_SV, TB5_SV, TB6_SV: REAL := 0;
	T_P2P_EN: TON := (PT:=T#10S);//통신 가능 -> TB MC 켜지고 TB 초기활 될때 까지 기다림. 이유 SMC TB가 전원이 새로 켜지면 SV를 읽어버린는 현상이 있음
	
	T_TMOut: TON := (PT:=T#1S);
	iStep: INT := 1;
	bTx_en: BOOL;
	bTx_ok: BOOL;
	bSV_mode: BOOL;
	addrMin: INT := 1;
	addrMax: INT := 6;
	
	//For Send
	T_Tx: TON := (PT:=T#10MS);
	fbTx: SendString;
	strTx: STRING;
	strTx_TEST: STRING;
	bTx_busy: BOOL;
	eTx_errID: ComError_t;	
		
	//For Receive
	T_Rx: TON := (PT:=T#10MS);
	bRx_ok: BOOL;	
	fbRx: ReceiveString;
	strRx: STRING;
	bRx_received: BOOL;
	bRx_busy: BOOL;
	eRx_errID: ComError_t;
	bRx_tmout: BOOL;
	strPV: STRING;

	iPvDecimal: INT := 1;// Config Data			
END_VAR

//TB: Thermal Bath x 6EA
//Maker: SMC
//Model: HEBC002-WA10
//Temp Range: -15 ~60℃
//RS485: 9600, DataBit(8), Parity(None), StopBit(1)
//BCC Check X

T_P2P_EN(IN:= do_TB_MC);

IF T_P2P_EN.Q AND bTx_en = Off THEN
	bTx_en := 1;
	bTx_ok := bRx_ok := 0;
	bSV_mode := 0;
	CASE iStep OF
	1:
	 IF TB1_SV <> sv_TB1 OR is_TB1_485_err THEN
		 TB1_SV := sv_TB1;
		 strTx := CONCAT(CONCAT('$0201WSV1', F_TB_SV2STR(TB1_SV)), '$03'); //TB1 SV Send
		 strTx_TEST := strTx;
		 bSV_mode := 1;
	 ELSE
		 strTx := '$0201RPV1$03'; //TB1 PV Req 
	 END_IF	
	2:
	 IF TB2_SV <> sv_TB2 OR is_TB2_485_err THEN
		 TB2_SV := sv_TB2;
		 strTx := CONCAT(CONCAT('$0202WSV1', F_TB_SV2STR(TB2_SV)), '$03'); //TB2 SV Send
		 bSV_mode := 1;
	 ELSE
		 strTx := '$0202RPV1$03'; //TB2 PV Req
	 END_IF
	3:
	 IF TB3_SV <> sv_TB3 OR is_TB3_485_err THEN
		 TB3_SV := sv_TB3;
		 strTx := CONCAT(CONCAT('$0203WSV1', F_TB_SV2STR(TB3_SV)), '$03'); //TB3 SV Send
		 bSV_mode := 1;
	 ELSE
		 strTx := '$0203RPV1$03'; //TB3 PV Req		
	 END_IF
	4:
	 IF TB4_SV <> sv_TB4 OR is_TB4_485_err THEN
		 TB4_SV := sv_TB4;
		 strTx := CONCAT(CONCAT('$0204WSV1', F_TB_SV2STR(TB4_SV)), '$03'); //TB4 SV Send
		 bSV_mode := 1;
	 ELSE
		 strTx := '$0204RPV1$03'; //TB4 PV Req		 
	 END_IF
	5:
	 IF TB5_SV <> sv_TB5 OR is_TB5_485_err THEN
		 TB5_SV := sv_TB5;
		 strTx := CONCAT(CONCAT('$0205WSV1', F_TB_SV2STR(TB5_SV)), '$03'); //TB5 SV Send
		 bSV_mode := 1;
	 ELSE
		 strTx := '$0205RPV1$03'; //TB5 PV Req		 
	 END_IF
	6:
	 IF TB6_SV <> sv_TB6 OR is_TB6_485_err THEN
		 TB6_SV := sv_TB6;
		 strTx := CONCAT(CONCAT('$0206WSV1', F_TB_SV2STR(TB6_SV)), '$03'); //TB6 SV Send
		 bSV_mode := 1;
	 ELSE
		 strTx := '$0206RPV1$03'; //TB6 PV Req		 
	 END_IF	
	END_CASE;
	
END_IF;


//Tx
T_Tx(IN:=bTx_en AND bTx_ok = 0 );
IF T_Tx.Q OR fbTx.Busy THEN
	bTx_ok := 1;	
	fbTx(SendString:= strTx, TXbuffer:= TxBuf_TB, Busy=> bTx_busy, Error=> );	
	IF fbTx.Error <> COMERROR_NOERROR THEN
		eTx_errID := fbTx.Error;
		bTx_ok := 0;
	ELSE
		eTx_errID := COMERROR_NOERROR;
		bTx_ok := 1;					
	END_IF;
END_IF;

//Rx
fbRx(Prefix:= '$02', Suffix:= '$03',
	Timeout:= T#1S, ReceivedString:= strRx,
	RXbuffer:= RxBuf_TB, StringReceived=> bRx_received,
	Busy=> bRx_busy, Error=> eRx_errID,
	RxTimeout=> bRx_tmout);
	
IF bRx_received THEN
	bRx_received := 0;
	bRx_ok := 1;	
	
	IF bSV_mode THEN//Write SV				
		strPV := MID(STR:=strRx, LEN:=1, POS:=4); //'$06' TB:'$0201$06$03'
		IF strPV = '$06' THEN
			CASE iStep OF
				1: 	is_TB1_485_err := 0;
				2:	is_TB2_485_err := 0;
				3:	is_TB3_485_err := 0;
				4:	is_TB4_485_err := 0;
				5:	is_TB5_485_err := 0;
				6:	is_TB6_485_err := 0;
			END_CASE;	
		END_IF;
	ELSE//Read PV						
		strPV := MID(STR:=strRx, LEN:=5, POS:=8); //TB:'$0201$06PV100250$03'
		IF strPV = 'HHHHH' THEN
			CASE iStep OF
				1: 	pv_TB1 := -1.0; is_TB1_TC_bk := 1; is_TB1_485_err := 0;
				2:	pv_TB2 := -1.0; is_TB2_TC_bk := 1; is_TB2_485_err := 0;
				3:	pv_TB3 := -1.0; is_TB3_TC_bk := 1; is_TB3_485_err := 0;
				4:	pv_TB4 := -1.0; is_TB4_TC_bk := 1; is_TB4_485_err := 0;
				5:	pv_TB5 := -1.0; is_TB5_TC_bk := 1; is_TB5_485_err := 0;
				6:	pv_TB6 := -1.0; is_TB6_TC_bk := 1; is_TB6_485_err := 0;
			END_CASE;	
		ELSE
			CASE iStep OF
				1: 	pv_TB1 := F_TB_PV2REAL(strPV); is_TB1_TC_bk := 0; is_TB1_485_err := 0;      //F_LH_PV(hexPV:= strPV, nDecimal:= iPvDecimal);
				2:	pv_TB2 := F_TB_PV2REAL(strPV); is_TB2_TC_bk := 0; is_TB2_485_err := 0;
				3:	pv_TB3 := F_TB_PV2REAL(strPV); is_TB3_TC_bk := 0; is_TB3_485_err := 0;
				4:	pv_TB4 := F_TB_PV2REAL(strPV); is_TB4_TC_bk := 0; is_TB4_485_err := 0;
				5:	pv_TB5 := F_TB_PV2REAL(strPV); is_TB5_TC_bk := 0; is_TB5_485_err := 0;
				6:	pv_TB6 := F_TB_PV2REAL(strPV); is_TB6_TC_bk := 0; is_TB6_485_err := 0;
			END_CASE;
		END_IF;
	END_IF;	
END_IF;
	
//Next TB
//addrMax := 6;
T_Rx(IN:= bRx_ok);
T_TMOut(IN:= bRx_received = 0);
IF T_Rx.Q OR T_TMOut.Q THEN
	T_Rx(IN:= 0);	
	bTx_en := 0;
	
	IF T_TMOut.Q THEN //TimeOut Error Check
		CASE iStep OF
		1: 	is_TB1_485_err := 1;
		2:	is_TB2_485_err := 1;
		3:	is_TB3_485_err := 1;
		4:	is_TB4_485_err := 1;
		5:	is_TB5_485_err := 1;
		6:	is_TB6_485_err := 1;
		END_CASE;	
	END_IF;
	T_TMOut(IN:= 0);
	
	IF iStep < addrMax THEN	
		iStep := iStep + 1;
	ELSE					
		iStep := addrMin; 
	END_IF;
END_IF;

END_PROGRAM

// ---- POUs/MR_PRG/P11_Rx_TV.TcPOU
PROGRAM P11_Rx_TV
VAR
	Resolution: REAL := 32767;//0~7FFF	
	Resolution_CDG: REAL := 24576;//0~6000h
END_VAR

//Throttle Valve
pv_POS := WORD_TO_REAL(Rx_TV_POS) * N_MAX[28] / Resolution; //TV POS
pv_P01 := WORD_TO_REAL(Rx_TV_CDG1) * N_MAX[29] / Resolution_CDG;//P01

//OP 상태 표시 
ing_TV_presCtrl := (Rx_TV_ST = 0);
ing_TV_posCtrl := (Rx_TV_ST = 1);
is_TV_open := (Rx_TV_ST = 2);
is_TV_init_X := (Rx_TV_ST = 3);
is_TV_close := (Rx_TV_ST = 4);
is_TV_fail := (Rx_TV_ST = 5);
ing_TV_init := (Rx_TV_ST = 6);
is_TV_stop := Tx_TV_Mode <> 0 AND (Rx_TV_ST = 8);
is_TV_run := Tx_TV_Mode = 0;//ing_TV_presCtrl OR ing_TV_posCtrl;

END_PROGRAM

// ---- POUs/MR_PRG/P12_Rx_IH.TcPOU
PROGRAM P12_Rx_IH
VAR
	r1: REAL;
END_VAR

//Induction Heater Controller : E3508 
r1 := WORD_TO_REAL(Rx_IH_PV);

pv_IH := r1 / 10;

